# B&R Automation Studio project CombinedLinenCleanA6 (part 2)

#### picd.var
```iecst
VAR
	STEP : UINT;
END_VAR
VAR RETAIN
	PLS : BOOL;
	LASTSTEP : UINT;
END_VAR
VAR
	O_RunMotor : BOOL;
	I_OutgoingFull : BOOL;
	O_OpenSeparator : BOOL;
	ReleasedToIncline : BOOL;
	ReleasedToInclineET : TIME;
	NoBags : BOOL;
	StopInclineET : TIME;
	StopIncline : BOOL;
	I_PaddleInPosition : BOOL;
	BagArriveIncline : BOOL;
	I_ArriveIncline : BOOL;
	TransitWindowClosedET : TIME;
	TransitWindowClosed : BOOL;
	BagReleasedSep : BOOL;
	I_BagAtSep : BOOL;
	I_TrolleyOutAtBott : BOOL;
	I_TrolleyOnIncline : BOOL;
	BagReleased : BOOL;
	mySeq : UINT;
	myIO : UINT;
	myBufferBag : UINT;
	myRelLine : UINT;
	myLine : UINT;
	myLastBag : UINT;
	myFirstBag : UINT;
	myX20IO : UINT;
	I_BagReleasedSep : BOOL;
	TimerAlarm : TON_10ms;
	myRelBag : UINT;
	myIC : UINT;
	DestValid : BOOL;
	myZone : INT;
	SettledAtSep : BOOL;
	SettledAtSepET : UDINT;
	I_BagInSep : BOOL;
	SettledInSep : BOOL;
	SettledInSepET : UDINT;
	BagArrived : BOOL;
END_VAR
```

### Program Logical/Reference/36_picu7 (IEC) - *PICU7 Incline up Empty trolleys

#### picu.ab
```automation-basic
PROGRAM _CYCLIC
	(* cyclic program *)

;Sequence 30 - Primary Incline Conveyor 4 D[900 + mySeq]

;-----------------------------------------
;Revision 1.00 17/04/2007 D.J. First Issue
;-----------------------------------------
mySeq 	= 36
myIO	= 177
myZone	= 0

I_PaddleInPosition		= X[myIO].X01
I_BagAtSep              = X[myIO].X03
I_BagArriveIncline		= X[myIO].X04
I_OutgoingFull			= X[myIO].X05

O_RunMotor 				= FALSE
O_OpenSeparator			= FALSE

;Setup Sequence
;-----------------------
STEP = D[900 + mySeq]
;Setup Pulse contact
PLS = (STEP <> LASTSTEP)
LASTSTEP = STEP

;If no bags on the buffers then stop the motor
NoBags = (STEP = 1) AND NOT I_BagAtSep
TON_10ms(NoBags,2000,StopIncline,StopInclineET)
TON_10ms(I_OutgoingFull,100,OutgoingFull,OutgoingFullET)

O_RunMotor = (NOT OutgoingFull AND NOT StopIncline AND NOT Std.HaltSysZone[myZone] AND (STEP <> 0) AND (STEP <> 2)); AND (STEP <> 2))

IF (STEP = 0) THEN
;	D[900 + mySeq] = 1
ENDIF

;Run Incline until paddle in position
IF (STEP = 1) THEN
	IF (I_PaddleInPosition AND I_BagAtSep AND O_RunMotor) THEN
		D[900 + mySeq] = 2
	ENDIF
ENDIF

;Open Separator 1.5 seconds
;Allow 3 sec for trolley to be detected releasing from separator
TON_10ms((STEP = 2),150,ReleasedToIncline,ReleasedToInclineET)
TON_10ms(ReleasedToIncline,550,TransitWindowClosed,TransitWindowClosedET)
IF (STEP = 2) THEN
	O_OpenSeparator	= NOT ReleasedToIncline
	IF I_BagArriveIncline OR TransitWindowClosed THEN
		D[900 + mySeq] = 3
	ENDIF
	ELSE
	ReleasedToIncline = FALSE
ENDIF

;Check not stpped on paddle
IF (STEP = 3) THEN
	IF NOT I_PaddleInPosition THEN
		D[900 + mySeq] = 1
	ENDIF
ENDIF

Y[34].Y02		= O_RunMotor
Y[myIO].Y06 	= O_OpenSeparator
END_PROGRAM
```

### Program Logical/Reference/38_picu9 (IEC) - *PICU9 Incline up Empty trolleys

#### picu.ab
```automation-basic
PROGRAM _CYCLIC
	(* cyclic program *)

;Sequence 30 - Primary Incline Conveyor 4 D[900 + mySeq]

;-----------------------------------------
;Revision 1.00 17/04/2007 D.J. First Issue
;-----------------------------------------
mySeq 	= 38
myIO	= 179
myZone	= 0

I_PaddleInPosition		= X[myIO].X01
I_BagAtSep              = X[myIO].X03
I_BagArriveIncline		= X[myIO].X04
I_OutgoingFull			= X[myIO].X05

O_RunMotor 				= FALSE
O_OpenSeparator			= FALSE

;Setup Sequence
;-----------------------
STEP = D[900 + mySeq]
;Setup Pulse contact
PLS = (STEP <> LASTSTEP)
LASTSTEP = STEP

;If no bags on the buffers then stop the motor
NoBags = (STEP = 1) AND NOT I_BagAtSep
TON_10ms(NoBags,750,StopIncline,StopInclineET)
TON_10ms(I_OutgoingFull,100,OutgoingFull,OutgoingFullET)

O_RunMotor = (NOT OutgoingFull AND NOT StopIncline AND NOT Std.HaltSysZone[myZone] AND (STEP <> 0) AND (STEP <> 2))

IF (STEP = 0) THEN
	D[900 + mySeq] = 1
ENDIF

;Run Incline until paddle in position
IF (STEP = 1) THEN
	IF (I_PaddleInPosition AND I_BagAtSep AND O_RunMotor) THEN
		D[900 + mySeq] = 2
	ENDIF
ENDIF

;Open Separator 1.5 seconds
;Allow 3 sec for trolley to be detected releasing from separator
TON_10ms((STEP = 2),150,ReleasedToIncline,ReleasedToInclineET)
TON_10ms(ReleasedToIncline,550,TransitWindowClosed,TransitWindowClosedET)
IF (STEP = 2) THEN
	O_OpenSeparator	= NOT ReleasedToIncline
	IF TransitWindowClosed OR I_BagArriveIncline THEN
		D[900 + mySeq] = 3
	ENDIF
	ELSE
	ReleasedToIncline = FALSE
ENDIF

;Check not stpped on paddle
IF (STEP = 3) THEN
	IF NOT I_PaddleInPosition THEN
		D[900 + mySeq] = 1
	ENDIF
ENDIF

Y[34].Y04 		= O_RunMotor
Y[myIO].Y06 	= O_OpenSeparator
END_PROGRAM
```

### Program Logical/Reference/39_picu10 (IEC) - *PICU10 Incline up Empty trolleys

#### picu.ab
```automation-basic
PROGRAM _CYCLIC
	(* cyclic program *)

;Sequence 30 - Primary Incline Conveyor 4 D[900 + mySeq]

;-----------------------------------------
;Revision 1.00 17/04/2007 D.J. First Issue
;-----------------------------------------
mySeq 	= 39
myIO	= 180
myZone	= 2

I_PaddleInPosition		= X[myIO].X01
I_BagAtSep              = X[myIO].X03
I_BagArriveIncline		= X[myIO].X04
I_OutgoingFull			= X[myIO].X05

O_RunMotor 				= FALSE
O_OpenSeparator			= FALSE

;Setup Sequence
;-----------------------
STEP = D[900 + mySeq]
;Setup Pulse contact
PLS = (STEP <> LASTSTEP)
LASTSTEP = STEP

;If no bags on the buffers then stop the motor
NoBags = (STEP = 1) AND NOT I_BagAtSep
TON_10ms(NoBags,3000,StopIncline,StopInclineET)
TON_10ms(I_OutgoingFull,100,OutgoingFull,OutgoingFullET)

O_RunMotor = (NOT OutgoingFull AND NOT StopIncline AND NOT Std.HaltSysZone[myZone] AND (STEP <> 0) AND (STEP <> 2))

IF (STEP = 0) THEN
	;D[900 + mySeq] = 1
ENDIF

;Run Incline until paddle in position
IF (STEP = 1) THEN
	IF (I_PaddleInPosition AND I_BagAtSep AND O_RunMotor) THEN
		D[900 + mySeq] = 2
	ENDIF
ENDIF

;Open Separator 1.5 seconds
;Allow 3 sec for trolley to be detected releasing from separator
TON_10ms((STEP = 2),150,ReleasedToIncline,ReleasedToInclineET)
TON_10ms(ReleasedToIncline,550,TransitWindowClosed,TransitWindowClosedET)
IF (STEP = 2) THEN
	O_OpenSeparator	= NOT ReleasedToIncline
	IF TransitWindowClosed OR I_BagArriveIncline THEN
		D[900 + mySeq] = 3
	ENDIF
	ELSE
	ReleasedToIncline = FALSE
ENDIF

;Check not stpped on paddle
IF (STEP = 3) THEN
	IF NOT I_PaddleInPosition THEN
		D[900 + mySeq] = 1
	ENDIF
ENDIF

Y[34].Y05 		= O_RunMotor
Y[myIO].Y06 	= O_OpenSeparator
END_PROGRAM
```

### Program Logical/Reference/42_picd13 (IEC) - *PICU13 Incline down Empty trolleys

#### picu.ab
```automation-basic
PROGRAM _CYCLIC
	(* cyclic program *)

;Sequence 30 - Primary Incline Conveyor 4 D[900 + mySeq]

;-----------------------------------------
;Revision 1.00 17/04/2007 D.J. First Issue
;-----------------------------------------
mySeq 	= 42
myIO	= 183
myZone	= 3

I_PaddleInPosition		= X[myIO].X01
I_BagAtSep              = X[myIO].X03
I_BagArriveIncline		= X[myIO].X04
I_OutgoingFull			= X[myIO].X05

O_RunMotor 				= FALSE
O_OpenSeparator			= FALSE

;Setup Sequence
;-----------------------
STEP = D[900 + mySeq]
;Setup Pulse contact
PLS = (STEP <> LASTSTEP)
LASTSTEP = STEP

;If no bags on the buffers then stop the motor
NoBags = (STEP = 1) AND NOT I_BagAtSep
TON_10ms(NoBags,2000,StopIncline,StopInclineET)
TON_10ms(I_OutgoingFull,100,OutgoingFull,OutgoingFullET)

O_RunMotor = (NOT OutgoingFull AND NOT StopIncline AND NOT Std.HaltSysZone[myZone] AND (STEP <> 2))

IF (STEP = 0) THEN
	D[900 + mySeq] = 1
ENDIF

;Run Incline until paddle in position
IF (STEP = 1) THEN
	IF (I_PaddleInPosition AND I_BagAtSep AND O_RunMotor) THEN
		D[900 + mySeq] = 2
	ENDIF
ENDIF

;Open Separator 1.5 seconds
;Allow 3 sec for trolley to be detected releasing from separator
TON_10ms((STEP = 2),150,ReleasedToIncline,ReleasedToInclineET)
TON_10ms(ReleasedToIncline,550,TransitWindowClosed,TransitWindowClosedET)
IF (STEP = 2) THEN
	O_OpenSeparator	= NOT ReleasedToIncline
	IF TransitWindowClosed OR I_BagArriveIncline THEN
		D[900 + mySeq] = 3
	ENDIF
	ELSE
	ReleasedToIncline = FALSE
ENDIF

;Check not stpped on paddle
IF (STEP = 3) THEN
	IF NOT I_PaddleInPosition THEN
		D[900 + mySeq] = 1
	ENDIF
ENDIF

Y[23].Y04 		= O_RunMotor
Y[myIO].Y06 	= O_OpenSeparator
END_PROGRAM
```

### Program Logical/Reference/44_picd15 (IEC) - *PICU15 Incline down Empty trolleys

#### picu.ab
```automation-basic
PROGRAM _CYCLIC
	(* cyclic program *)

;Sequence 30 - Primary Incline Conveyor 4 D[900 + mySeq]

;-----------------------------------------
;Revision 1.00 17/04/2007 D.J. First Issue
;-----------------------------------------
mySeq 	= 44
myIO	= 185
myZone	= 3

I_PaddleInPosition		= X[myIO].X01
I_BagAtSep              = X[myIO].X03
I_BagArriveIncline		= X[myIO].X04
I_OutgoingFull			= X[myIO].X05

O_RunMotor 				= FALSE
O_OpenSeparator			= FALSE

;Setup Sequence
;-----------------------
STEP = D[900 + mySeq]
;Setup Pulse contact
PLS = (STEP <> LASTSTEP)
LASTSTEP = STEP

;If no bags on the buffers then stop the motor
NoBags = (STEP = 1) AND NOT I_BagAtSep
TON_10ms(NoBags,2000,StopIncline,StopInclineET)
TON_10ms(I_OutgoingFull,100,OutgoingFull,OutgoingFullET)

O_RunMotor = (NOT OutgoingFull AND NOT StopIncline AND NOT Std.HaltSysZone[myZone] AND (STEP <> 2))

IF (STEP = 0) THEN
	D[900 + mySeq] = 1
ENDIF

;Run Incline until paddle in position
IF (STEP = 1) THEN
	IF (I_PaddleInPosition AND I_BagAtSep AND O_RunMotor) THEN
		D[900 + mySeq] = 2
	ENDIF
ENDIF

;Open Separator 1.5 seconds
;Allow 3 sec for trolley to be detected releasing from separator
TON_10ms((STEP = 2),150,ReleasedToIncline,ReleasedToInclineET)
TON_10ms(ReleasedToIncline,550,TransitWindowClosed,TransitWindowClosedET)
IF (STEP = 2) THEN
	O_OpenSeparator	= NOT ReleasedToIncline
	IF TransitWindowClosed OR I_BagArriveIncline THEN
		D[900 + mySeq] = 3
	ENDIF
	ELSE
	ReleasedToIncline = FALSE
ENDIF

;Check not stpped on paddle
IF (STEP = 3) THEN
	IF NOT I_PaddleInPosition THEN
		D[900 + mySeq] = 1
	ENDIF
ENDIF

Y[23].Y06 		= O_RunMotor
Y[myIO].Y06 	= O_OpenSeparator
END_PROGRAM
```

### Program Logical/Reference/48_49_fbppr (IEC) - *Full bag pressure reliefs buffers before PUPs

#### fb_pr.var
```iecst
VAR CONSTANT
	Dec_C_MaxPressureReliefs : UINT := 2;
END_VAR
VAR RETAIN
	LASTSTEP : ARRAY[0..Dec_C_MaxPressureReliefs] OF UINT;
END_VAR
VAR
	PLS : ARRAY[0..Dec_C_MaxPressureReliefs] OF BOOL;
	STEP : UINT;
	TimerAlarm : ARRAY[0..Dec_C_MaxPressureReliefs] OF TON_10ms;
	mySeq : UINT;
	I_BagAtPR : ARRAY[0..Dec_C_MaxPressureReliefs] OF BOOL;
	n : INT;
	BagSettled : ARRAY[0..Dec_C_MaxPressureReliefs] OF TON_10ms;
	myRelLine : UINT;
	myLastBag : UINT;
	myBag : UINT;
	O_OpenStop : ARRAY[0..Dec_C_MaxPressureReliefs] OF BOOL;
	myOutLine : ARRAY[0..Dec_C_MaxPressureReliefs] OF USINT;
	I_BagReleased : ARRAY[0..Dec_C_MaxPressureReliefs] OF BOOL;
	BagReleased : ARRAY[0..Dec_C_MaxPressureReliefs] OF BOOL;
	myLine : ARRAY[0..Dec_C_MaxPressureReliefs] OF USINT;
	myZone : INT;
	I_BagInSep : ARRAY[0..3] OF BOOL;
	SettledInSep : ARRAY[0..3] OF TON_10ms;
	x : UINT;
	TestIndex : UINT;
	ReleaseValid : ARRAY[0..4] OF BOOL;
END_VAR
```

### Package Logical/Sequences - *GCS Primary 

- Program Logical/Sequences/10ms/zzPrimSearch (IEC) - *Search for ongoing lines using SLAC looking at last bag in transit (no source held here)

### Program Logical/Sequences/10ms/zzStnSer (IEC, version 2.00.0)

#### zzstnser.ab
```automation-basic
;-----------------------------------------------------
;Sorting Station Search Routine - No changes required!
;-----------------------------------------------------

;----------------------------------------
;Version 1.00 19/12/2005 First Issue D.J.
;Version 2.00 03/11/2010 Revised D.J.
;----------------------------------------

PROGRAM _CYCLIC

;Only one Bank / Loading VC can search in a given scan.

Bank = Bank + 1
IF (Bank > Std.MaxStationBanks) THEN
	Bank = 1
ENDIF

;Clear Array
Std.StnsToPurge = FALSE
LOOP n = 0 TO Std.MaxWeighstations DO
	;IF Stn[n].Purge THEN
	;	Std.StnsToPurge = TRUE
	;ENDIF
	BagInList[n] = FALSE
	SearchBagArray[n] = 0
ENDLOOP
TON_10ms(Std.StnsToPurge,100,StartPurge,StartPurgeET) ; use a timer to wait for all purge events to be recieved from trackview

MixCats			= (D[369] > 0)
MixCusts		= (D[366] > 0)	;Allow mixing of customers?
MixProgs		= (D[367] > 0)	;Allow mixing of Programs?

IF MixProgs	 THEN					;IF mixing programs then type must be mixed also.....
	D[368] =  1
ENDIF
MixProgTyp			= (D[368] > 0) 	;Allow mixing of Program Types?

;IF Std.ReversingBelt THEN
;	MaxReverseWeight	= D[370]			;Max weight to reverse..
;ELSE
	;MaxReverseWeight = 0
;ENDIF
;Send Status to Trackview -- BitWise OR to look at all banks

;PurgeOn = (Std.PurgeBank[1].PurgeOn OR Std.PurgeBank[2].PurgeOn OR Std.PurgeBank[3].PurgeOn OR Std.PurgeBank[4].PurgeOn)
;StatusReg = (Std.PurgeBank[1].StationsStatus OR Std.PurgeBank[2].StationsStatus OR Std.PurgeBank[3].StationsStatus OR Std.PurgeBank[4].StationsStatus)
D[360] = PurgeOn
memcpy(ADR(D[371]),ADR(StatusReg),4)
;Used by other sequences that need to check for Line[x].SpaceBIT direct
;eg. Loading VC will look for Enable.Search = 3
Enable.Search = Bank

IF (Bank <= Std.MaxStationBanks) THEN

	IF (Ldg[Bank].Search = 1) THEN

		Ldg[Bank].Found = 0
		Ldg[Bank].Line  = 0

		SearchFound = 0
		SearchLine  = 0

		Stn[0].QTime = 0

		LOOP x = Ldg[Bank].StartStn TO Ldg[Bank].EndStn DO
		;	x = 11
			n = x
			;Std.StnsToPurge = TRUE    ;KEV

			IF (Std.StnsToPurge AND Std.Purging) THEN	;Search through purge Stations to find bags that can be mixed

				IF Bank = 1 THEN
					Break
;					IF NOT TestTim THEN
;						GOTO Debug
;					ENDIF
				ELSE IF Bank = 2 THEN
					Break
				ENDIF
				;Purge doesn;t need to be in x loop so exit if > 1
				EXITIF x > Ldg[Bank].StartStn
				IF StartPurge THEN
					PurgeBatchSize	= 0
					BatchFound = FALSE
					; 1st put all bags to be searched into an array to reduce scanning through all stations bags
					LOOP r = 0 TO Std.MaxWeighstations DO
				;		Std.PurgeBank[Bank].PurgeBatch[r] = 0
					;	IF Stn[r].Purge AND (Stn[r].Weight > 0) AND NOT BagInList[r] AND (r >= Ldg[Bank].StartStn) AND (r <= Ldg[Bank].EndStn)  THEN
				;			SearchBagArray[Std.MaxWeighstations] = Std.StationBagsStart[Bank] + (r-Ldg[Bank].StartStn)
				;			BagInList[r] = TRUE
					;	ENDIF
						;Shuffle array
						LOOP s = Std.MaxWeighstations DOWNTO 1 DO
							IF (SearchBagArray[s-1] = 0) AND (SearchBagArray[s] > 0) THEN
								SearchBagArray[s-1] = SearchBagArray[s]
								SearchBagArray[s] = 0
								EndofBagArray = (s - 1)
							ENDIF
						ENDLOOP
					ENDLOOP
					;LOOP r = 0 TO EndofBagArray DO ; Start Searching through bags
					r = 0 ;Only search through from 1st bag in array as we already know it is to purge
					ReSearch = FALSE
					MisMatchedLoad = FALSE
					SearchIndex = 0
					StartSearch: ;Marker to re-search
					IF ReSearch THEN
						r = SearchIndex
					ENDIF
					LOOP s = 0 TO Std.MaxWeighstations DO
						PurgeBags[s] = 0
					ENDLOOP
					LOOP s = EndofBagArray DOWNTO 0 DO
						myBag_n = SearchBagArray[r]
						myBag_x = SearchBagArray[s]
						MatchCust = FALSE
						MatchCat = FALSE
						MatchProgType = FALSE
						MatchProg = FALSE
						BankValid = TRUE;((myBag_n >= Ldg[Bank].StartStn) AND (myBag_n <= Ldg[Bank].EndStn) AND (myBag_x >= Ldg[Bank].StartStn) AND (myBag_x <= Ldg[0].EndStn))

						;Check customer 1st
						IF (Bag[myBag_n].Cus = Bag[myBag_x].Cus) OR MixCusts THEN
							MatchCust = TRUE
						ENDIF
						IF (Bag[myBag_n].Cat = Bag[myBag_x].Cat) OR MixCats	 THEN
							MatchCat = TRUE
						ENDIF
					;	IF (Bag[myBag_n].Prg = Bag[myBag_x].Prg) OR MixProgs THEN
					;		MatchProg = TRUE
					;	ENDIF
					;	IF (D[2900 + Bag[myBag_n].Prg] = D[2900 + Bag[myBag_x].Prg]) OR MixProgTyp THEN
					;		MatchProgType = TRUE
					;	ENDIF

						MatchBags = (MatchCust AND MatchCat AND MatchProg AND MatchProgType AND BankValid)
						IF MatchBags THEN ; Put bag into another array so they can be best matched by weight
							;PurgeBags[0] = myBag_n
							PurgeBags[Std.MaxWeighstations] = myBag_x
							LOOP t = Std.MaxWeighstations DOWNTO 1 DO
								IF (PurgeBags[t] > 0) AND (PurgeBags[t-1] = 0) THEN
									PurgeBags[t -1] = PurgeBags[t]
									PurgeBags[t] = 0
									PurgeBatchSize	= t
								ENDIF
							ENDLOOP
						ENDIF
					ENDLOOP ; Ony research if no matching bags, and the bag searched is to small for a batch
					IF ((PurgeBatchSize = 1) AND (Bag[PurgeBags[0]].Wgt < MaxReverseWeight)) THEN
						ReSearch = TRUE
						INC SearchIndex
						;Check when all bags have been searched...
						IF (SearchBagArray[SearchIndex] = 0) THEN
							;INC SearchIndex
							;The only bags left cannot be put in the same bag and should be classified as a mixed load.
							MisMatchedLoad = (SearchIndex > 1)
							LOOP y = 0 TO SearchIndex - 1 DO
								PurgeBags[y] = 	SearchBagArray[y]
							ENDLOOP
							PurgeBatchSize = SearchIndex
						ELSE
							GOTO StartSearch
						ENDIF
					ENDIF

					;ENDLOOP
					;Matching bags are in the array Purge Bags. Try to fit into a load?
					;Bag 0 in the array is that master.. This is the data that will go into a bag.. so we will get the batch weight from this program code.
					;Put all bag into wieght order highest first..
					LOOP r = 0 TO 19 DO
						BagInList[r] = FALSE
						PurgeBagsInWgtOrder[r] = 0
					ENDLOOP
					IF (PurgeBatchSize > 0) THEN
						GetStn =  ((PurgeBags[0] - Std.StationBagsStart[Bank]) + 1)
						IF (GetStn < Std.MaxWeighstations) THEN
							MaxBatchWieght = D[4900 + GetStn] ;SP3
						ENDIF
						IF (MaxBatchWieght = 0) OR (MaxBatchWieght <= MaxReverseWeight) THEN
							 MaxBatchWieght = MaxReverseWeight + 100
						ENDIF

						LOOP r = 0 TO (PurgeBatchSize - 1) DO
							BagWgt = 0
							LOOP s = 0 TO (PurgeBatchSize - 1) DO
								IF (Bag[PurgeBags[s]].Wgt > 0) AND (Bag[PurgeBags[s]].Wgt > BagWgt) AND NOT BagInList[s] THEN
									BagWgt = Bag[PurgeBags[s]].Wgt
									BagNum = PurgeBags[s]
									Index = s
								ENDIF
							ENDLOOP
							PurgeBagsInWgtOrder[r] = USINT(BagNum)
							BagInList[Index] = TRUE
						ENDLOOP ;
						IF (MaxBatchWieght > MaxReverseWeight) AND (Bag[PurgeBagsInWgtOrder[0]].Wgt > 0)THEN ; Check no errors in batch sizes.. Reverse all loads if fault
							;Now bags are in weight order make the best by adding the highest values until bag is full
							BatchWeight = 0
							PurgeBagsQty = 0
							;IF (Bag[PurgeBagsInWgtOrder[0]].Wgt  < MaxBatchWieght) THEN
							BatchWeight = Bag[PurgeBagsInWgtOrder[0]].Wgt
							BatchCount = Bag[PurgeBagsInWgtOrder[0]].Cnt
						;	Std.PurgeBank[Bank].PurgeBatch[0] = PurgeBagsInWgtOrder[0]
							;ENDIF
							LOOP r = 1 TO PurgeBatchSize DO ; Start from 1 as index 0 is highest weight so always in the array
								myBag = PurgeBagsInWgtOrder[r]
								IF ((Bag[myBag].Wgt + BatchWeight) <= MaxBatchWieght) THEN
									BatchWeight = Bag[myBag].Wgt + BatchWeight
									BatchCount = Bag[myBag].Cnt + BatchCount
							;		Std.PurgeBank[Bank].PurgeBatch[PurgeBatchSize] = USINT(myBag)
									PurgeBagsQty = PurgeBagsQty + 1
								ENDIF
								;Shuffle down array
								LOOP s = PurgeBatchSize DOWNTO 1 DO
								;	IF (Std.PurgeBank[Bank].PurgeBatch[s] > 0) AND (Std.PurgeBank[Bank].PurgeBatch[s - 1] = 0) THEN
								;		Std.PurgeBank[Bank].PurgeBatch[s - 1] = Std.PurgeBank[Bank].PurgeBatch[s]
								;		Std.PurgeBank[Bank].PurgeBatch[s] = 0
								;	ENDIF
								ENDLOOP
							;	IF (r = PurgeBatchSize) AND (Std.PurgeBank[Bank].PurgeBatch[0] > 0) THEN
							;		BatchFound = TRUE
							;	ENDIF
							EXITIF BatchFound = TRUE
							ENDLOOP
						ENDIF
;					ELSE
;						GOTO ExitPurge ;Invalid purge..
					ENDIF
					IF BatchFound AND NOT MisMatchedLoad THEN ;Bags found;
						IF (BatchWeight >=  MaxReverseWeight) THEN ; Wieght it OK purge into Bag search for destination.

							IF NO THEN
								SearchFound  		= 99
								SearchLine   		= 0;LineSearch[Choice]
								Ldg[Bank].Search   	= 2
							ELSE	;
								;Check line choice 1st to 4th in order if any valid then exit loop
								;StnNum = (Std.PurgeBank[Bank].PurgeBatch[0] - (Std.StationBagsStart[Bank] - Ldg[Bank].StartStn)) ; Get station number from Bag number.
						;		StnCat =  Bag[Std.PurgeBank[Bank].PurgeBatch[0]].Prg

								LineSearch[1]   = D[3000 + StnCat]
								LineSearch[2]   = D[3100 + StnCat]
								LineSearch[3]   = D[3200 + StnCat]
								LineSearch[4]   = D[3300 + StnCat]

								LOOP Choice = 1 TO 4 DO
									LineValid = (D[20 + LineSearch[Choice]] > 0)
									IF (LineSearch[Choice] > 0) AND (Line[LineSearch[Choice]].SpaceBIT >= 1) AND LineValid THEN
										SearchFound  		= 99
										SearchLine   		= LineSearch[Choice]
										Ldg[Bank].Search   	= 2
									ENDIF
									EXITIF (SearchFound > 0)
								ENDLOOP
							ENDIF
						ELSE ; Load/s is to small reverse.

							SearchFound  		= 98
							SearchLine   		= 0
							Ldg[Bank].Search   	= 2
						ENDIF
					ELSE IF MisMatchedLoad THEN
						SearchFound  		= 97
						SearchLine   		= 0
						Ldg[Bank].Search   	= 2
					ENDIF
					IF SearchFound > 90 THEN ;If bags are found remove from purging Q
;						Std.PurgeBank[Bank].PurgeBagQty	= PurgeBagsQty

;						Std.PurgeBank[Bank].PurgeBatchWieght = BatchWeight
;					Std.PurgeBank[Bank].PurgeBatchCount	= BatchCount
;						LOOP r = 0 TO PurgeBagsQty - 1 DO
;							IF (Std.PurgeBank[Bank].PurgeBatch[r] > 0) THEN
;								StnNum = (Std.PurgeBank[Bank].PurgeBatch[r] - (Std.StationBagsStart[Bank] - Ldg[Bank].StartStn))
;								;Stn[StnNum].QTime = 0
;								;Stn[StnNum].Purge = FALSE
;							ENDIF
;						ENDLOOP
					ENDIF
				ENDIF
			ELSE IF ((Stn[n].QTime > 10) AND (Stn[n].QTime > Stn[0].QTime)) THEN

				;Destination has been given to bag by operator check
				LineSearchManual = Stn[n].DestManual

				IF Std.AutoLineAllocation THEN

					;Automatic Line Allocation - Line Space is never checked even if a destiantion has been edited
					SearchFound  		= n
					SearchLine   		= LineSearchManual
					Stn[0].QTime 		= Stn[n].QTime
					Ldg[Bank].Search   	= 2

				ELSE
					;1st 2nd 3rd and 4th Line choices
					LineSearch[1]   = D[4000 + n]
					LineSearch[2]   = D[4100 + n]
					LineSearch[3]   = D[4200 + n]
					LineSearch[4]   = D[4300 + n]

					;Always Search for at least 1 space
					IF (Stn[n].SpacesRequired = 0) THEN
						Stn[n].SpacesRequired = 1
					ENDIF

					;When manual is selected then the 1st 2nd 3rd and 4th are not checked
					IF (LineSearchManual > 0) THEN
						IF (Line[LineSearchManual].SpaceBIT > 0) THEN
							SearchFound  		= n
							SearchLine   		= LineSearchManual
							Stn[0].QTime 		= Stn[n].QTime
							Ldg[Bank].Search   	= 2
						ENDIF
					ELSE
							;Check line choice 1st to 4th in order if any valid then exit loop

						LOOP Choice = 1 TO 4 DO
							;Choice = 1
							LineValid = (D[20 + LineSearch[Choice]] > 0)
							IF (LineSearch[Choice] > 0) AND (Line[LineSearch[Choice]].SpaceBIT >= Stn[n].SpacesRequired) AND LineValid THEN
								SearchFound  		= n
								SearchLine   		= LineSearch[Choice]
								Stn[0].QTime 		= Stn[n].QTime
								Ldg[Bank].Search   	= 2

							ENDIF
							EXITIF (SearchFound > 0)
						ENDLOOP

					ENDIF

				ENDIF ;/AutoLineAllocation

			ENDIF

		ENDLOOP

		ExitPurge:
		IF (Ldg[Bank].Search = 2) THEN
			Ldg[Bank].Found  = SearchFound
			Ldg[Bank].Line   = SearchLine
		ELSE
			Ldg[Bank].Search = 0 ;Failed
		ENDIF

	ENDIF
ENDIF
Debug:

END_PROGRAM
```

### Program Logical/Sequences/10ms/zzCount (IEC) - Counting frames inputs & Piece Weights

#### zzcount.ab
```automation-basic
PROGRAM _CYCLIC
(* cyclic program *)

;Sorting station counting

CountMode 	= D[994]
CountOn		= (CountMode <> 0)
CountPiece 	= (CountMode = 1)
CountBoth	= (CountMode = 2)
CountCount	= (CountMode = 3)

Stn[1].CntInput 	= X[31].X01
Stn[2].CntInput 	= X[31].X02
Stn[3].CntInput 	= X[31].X03
Stn[4].CntInput 	= X[31].X04
Stn[5].CntInput 	= X[32].X01
Stn[6].CntInput 	= X[32].X02
Stn[7].CntInput 	= X[32].X03
Stn[8].CntInput 	= X[32].X04
Stn[9].CntInput 	= X[33].X01
Stn[10].CntInput 	= X[33].X02

LOOP n = 1 TO Std.MaxWeighstations DO

	;Get the category for the station
	StnCat = Bag[200 + n].Cat
	IF ((StnCat < 0) OR (StnCat > Std.MaxCats)) THEN
		StnCat = 0
	ENDIF

	;Read the Category database setting
	StnUsePiece		= (D[2900 + StnCat] > 0)
	StnPieceWgt		= (D[2800 + StnCat])
	;Set mode depending on loading program selection
	StnCountPiece 	= (CountPiece OR (CountBoth AND StnUsePiece))

	IF CountOn THEN
		;Count by input
		CountPLS[n].CLK = (Stn[n].CntInput AND NOT StnCountPiece)
		CountPLS[n] FUB R_TRIG()

		IF CountPLS[n].Q THEN
			Stn[n].Count = (Stn[n].Count + 1)
		ENDIF

		;Count by piece weight
		IF StnCountPiece THEN
			;Calculate the current count by piece weight
			StnGram = (Bag[200 + n].Wgt * 1000)
			IF (StnGram > 0) THEN
				IF (StnPieceWgt > 0) THEN
					;Calc Here
					Items = (StnGram / StnPieceWgt)
					;round up items
					Remainder = SINT(Items MOD 10)
					IF (Remainder > 4) THEN
						ItemsRound = (Items + 10)
					ELSE
						ItemsRound = Items
					ENDIF
					IF ((ItemsRound / 10) < 32767) THEN
						Stn[n].Count = UINT(ItemsRound / 10)
					ELSE
						Stn[n].Count = 32767
					ENDIF
				ELSE
					Stn[n].Count = 0
				ENDIF
			ELSE
				Stn[n].Count = 0
			ENDIF
		ENDIF
	ELSE
		Stn[n].Count = 0
	ENDIF

ENDLOOP

END_PROGRAM
```

### Program Logical/Sequences/10ms/zzStnMix (IEC) - * Station mixing Customer and Categories

#### zzstnmix.ab
```automation-basic
PROGRAM _CYCLIC
;----------------------
;Sorting Station Mixing
;----------------------

;----------------------------------------
;Version 1.00 09/12/2005 D.J. First Issue
;----------------------------------------

;Notes:
;When the operator changes either the Category or Customer of any station then the report should be written.
;If the Customer or Category is set to zero the report will be written for the previous Cat and Cus however
;the previous Cat and Cus will be set to zero. When the Cat or Cus is next changed there will be no report

IF Std.StationReports THEN

	;Special for Mewa only box 1 to 6 are reported on
	LOOP n = 1 TO Std.MaxWeighstations DO

		StnBag = n + (Std.StationBagsStart[1] - 1) ;Assumes all station bags will follow in order

		IF (ReportLoading[n].Cat = 0) THEN

			;Check if Category or Customer have been changed
			CatChanged 	= (Bag[StnBag].Cat <> StnPrev[n].Cat)
			CatValid   	= (StnPrev[n].Cat > 0)

			CusChanged 	= (Bag[StnBag].Cus <> StnPrev[n].Cus)
			CusValid   	= (StnPrev[n].Cus > 0)

			;Check if anything has been added and current weight is not less than the previous
			WgtValue 	= Stn[n].Weight	- INT(StnPrev[n].Wgt)
			WgtValid 	= (WgtValue > 0)

			;Check if anything has been added and current weight is not less than the previous
			CntValue 	= Stn[n].Count - INT(StnPrev[n].Cnt)
			CntValid 	= (CntValue > 0)

			;Ensure valid values as we report on either a weight or count change
			IF (WgtValue < 0) THEN
				WgtValue = 0
			ENDIF

			IF (CntValue < 0) THEN
				CntValue = 0
			ENDIF

			IF ((CatChanged OR CusChanged) AND CusValid AND CatValid AND (WgtValid OR CntValid)) THEN

				ReportLoading[n].Prg = StnPrev[n].Prg		;Program
				ReportLoading[n].Cat = StnPrev[n].Cat		;Category
				ReportLoading[n].Cus = StnPrev[n].Cus		;Customer
				ReportLoading[n].Wgt = UINT(WgtValue)		;Weight
				ReportLoading[n].Cnt = UINT(CntValue)		;Count
				ReportLoading[n].Stn = n         			;Station
				ReportLoading[n].Mcn = 0					;Machine
				ReportLoading[n].Bid = StnPrev[n].Bid		;Bag ID
				ReportLoading[n].Mis = n
				ReportLoading[n].Act = repMix
				ReportLoading[n].Ur1 = 0
				ReportLoading[n].Ur2 = 0
				ReportLoading[n].Rkg = 0

			ENDIF

			;Set Previous to Current even if the Previous values were not valid
			IF (CatChanged OR CusChanged) THEN
				StnPrev[n].Prg = Bag[StnBag].Prg
				StnPrev[n].Cat = Bag[StnBag].Cat
				StnPrev[n].Cus = Bag[StnBag].Cus
				StnPrev[n].Wgt = Stn[n].Weight
				StnPrev[n].Cnt = Stn[n].Count
				StnPrev[n].Bid = Bag[StnBag].Bid
			ENDIF

		ENDIF

	ENDLOOP

ENDIF

END_PROGRAM
```

### Program Logical/Sequences/10ms/zzStatus (IEC) - * System status

#### zzstatus.ab
```automation-basic
PROGRAM _CYCLIC
(* cyclic program *)

;System Status and Halting
;-------------------------

Std.StopSystem 				= (D[100] <> 0)

Std.EStop 					= NOT X[1].X01
Std.MotorOverload   		= NOT X[1].X02
Std.SafetyOn				= X[1].X03
Std.HaltSys					= NOT Std.SafetyOn ;OR Std.StopSystem)

Std.MaxZones 				= 1
Std.FireAlarm				= X[3].X01// ON when the fire alarm is healthy

Std.SafetyOnZone[0]		= Std.SafetyOn AND Std.FireAlarm
Std.SafetyOnZone[1]		= X[1].X03 AND Std.FireAlarm; Gated area for PIC 3,4,5,11 & PP3
Std.SafetyOnZone[2]		= FALSE; Area between belts on soiled pp12, PIC10
Std.SafetyOnZone[3]		= FALSE ;Loading Area
Std.SafetyOnZone[4]		= FALSE;Loading Area Gated + Upstairs storage

LOOP n = 0 TO Std.MaxZones DO
	Std.HaltSysZone[n]=  NOT Std.SafetyOnZone[n]
ENDLOOP

;Std.SafetyOnVC[30]			= TRUE
;Std.HaltSysVC[30]			= NOT Std.SafetyOnVC[30]
;
;Std.SafetyOnVC[2]			= TRUE
;Std.HaltSysVC[2]			= NOT Std.SafetyOnVC[2]

;set to TRUE if not required
LoadingStopped 	= TRUE ;(Bag[220].Prg = 0)
OngoingStopped 	= TRUE ;(Bag[224].Prg = 0)
OffgoingStopped = TRUE ;(Bag[225].Prg = 0)

;If no Bag In Transit and stop requested then set system to stopped D[100] = 2
IF Std.StopSystem THEN
	IF LoadingStopped AND OngoingStopped AND OffgoingStopped THEN
		D[100] = 2
	ENDIF
ENDIF

;Force I/O Enable - Max ? Minutes
ForceEnable = FALSE

tmrForce.IN = ForceEnable
tmrForce.PT = 90000 ;6000 = 1 Minute
tmrForce FUB TON_10ms()

IF ForceEnable AND NOT tmrForce.Q THEN
	D[319] = 1
ELSE
	D[319] = 0
ENDIF

END_PROGRAM
```

### Program Logical/Sequences/10ms/1_clu_1 (IEC, version 1.00.0) - * Loading unit SLU1

#### 3_slu_1Cyclic.ab
```automation-basic
PROGRAM _CYCLIC
	(* cyclic program *)

;--------------------------------
;Sequence 3 - Loading Unit D[903]
;--------------------------------

;Inputs / Ouputs

;Enable.TransferBelt[1]	= FALSE

//I_BagAtBuffer			= X[3].X10
I_BagFrontPast			= X[5].X13
I_BagInLoadingUnit		= X[5].X12
//I_BagOnCarriage         = X[5].X05

//I_ChuteBlocked			= X[3].X14
SwitchedOn			= (D[20] = 1)

O_MoveCompressorUp		= FALSE
O_MoveCompressorDn		= FALSE

O_OpenBufferStop		= FALSE
O_SteadyCylinders		= FALSE
O_OpenStop	 			= FALSE
CAN[1].BagReady         = FALSE

Enable.CVC[2]           = FALSE

O_OpenBufferStop2		= FALSE

Alarm[1].Name 		= 0
Alarm[1].Bag		= 31
Alarm[1].Beacon		= TRUE
Alarm[1].Extra	 	= 0
Alarm[1].Time		= 6000

;Setup Sequence
;--------------
STEP = D[901]
;Setup Pulse contact
PLS = (STEP <> LASTSTEP)
LASTSTEP = STEP

;Alarm
SwitchFault = ((STEP = 1) AND (I_BagFrontPast OR I_BagInLoadingUnit))
;TON_10ms(((NOT PLS) AND (SwitchFault) OR (STEP = 3) OR (STEP = 11)),3000,Alarm[51],AlarmET[51])

IF (STEP = 0) THEN
	;Disabled
ENDIF

;Check for no bag in loading unit
TON_10ms((NOT I_BagFrontPast AND NOT I_BagInLoadingUnit),200,TripsClear,TripsClearET)
IF (STEP = 1) THEN
	IF (NOT CAN[1].UnloadFinished AND SwitchedOn AND TripsClear) THEN
        D[901] = 2
	ENDIF
ENDIF

;Enable CVC2 to Send Bag
IF (STEP = 2) THEN
	Enable.CVC[2] = TRUE
	O_OpenStop	= TRUE
	IF I_BagFrontPast THEN
		D[901] = 3
   	ENDIF
ENDIF

;Bag Settles at loading unit
TON_10ms(I_BagInLoadingUnit,700,SettledAtStop,SettledAtStopET)
IF (STEP = 3) THEN
	Enable.CVC[2] = TRUE	;Must be on until bag is fully in the unit
	IF SettledAtStop THEN
		D[901] = 4
	ENDIF
	Alarm[1].Name = almBagNotArrived
	Alarm[1].Time		= 2000
ENDIF

;Steady bag
TON_10ms((STEP = 4),200,SteadysDown,SteadysDownET)
IF (STEP = 4) THEN
    IF SteadysDown THEN
		D[901] = 5
	ENDIF
ENDIF

;Steady cylinders on from steps 4 - 5
O_SteadyCylinders = ((STEP >= 4) AND (STEP <= 5))

;Move Steady Cylinders down
IF (STEP <> 5) THEN
	Cat 			= 0
	Cus			= 0
	kg			= 0
ENDIF

;Bag Ready to Driers
IF (STEP = 5) THEN
	IF PLS THEN
		Bag[31].Cat = 0
	ENDIF
	CAN[1].BagReady = TRUE
	IF CAN[1].UnloadFinished THEN
		FinishedLoading = TRUE
	ENDIF
	IF (CAN[1].Category > 0) THEN
		Cat 		= uint(CAN[1].Category)
		Cus			= uint(CAN[1].Customer)
		kg			= (CAN[1].Weight * 10)
	ENDIF
	IF FinishedLoading THEN
		Bag[31].Cat = usint(Cat)
		Bag[31].Cus	= Cus
		Bag[31].Wgt	= kg
		D[901] = 6
	ENDIF
ELSE
	FinishedLoading = FALSE
ENDIF

;Allow steadys to go up
TON_10ms((STEP = 6),200,SteadysUp,SteadysUpET)
IF (STEP = 6) THEN
    IF (SteadysUp  AND (Bag[31].Cat > 0))THEN
		D[901] = 7
	ENDIF
ENDIF

;Wait for Enable from CVC1
IF (STEP = 7) THEN
	IF Enable.CLU[1] THEN
		D[901] = 8
	ENDIF
ENDIF

;Release Bag
IF (STEP = 8) THEN
	O_OpenStop = TRUE
	IF NOT Enable.CLU[1] THEN
		D[901] = 1
	ENDIF
	Alarm[1].Name = almBagNotReleased
	Alarm[1].Time		= 2000
ENDIF

;Alarms
TimerAlarm.IN = NOT PLS AND (Alarm[1].Name > 0)
TimerAlarm.PT = Alarm[1].Time
TimerAlarm FUB TON_10ms()
Alarm[1].On = TimerAlarm.Q
Alarm[1].ET = TimerAlarm.ET
;Outputs
;-------

//Y[3].Y10 = O_OpenBufferStop
Y[5].Y12 = O_SteadyCylinders
Y[5].Y13 = O_OpenStop
;YM07 = O_OpenBufferStop2

//Y[3].Y13 = O_MoveCompressorDn

END_PROGRAM
```

#### 3_slu_1.var
```iecst
VAR RETAIN
	STEP : UINT;
	PLS : BOOL;
	LASTSTEP : UINT;
END_VAR
VAR
	EBagSettled : BOOL;
	EBagSettledET : TIME;
	O_OpenStop : BOOL;
	O_SteadyCylinders : BOOL;
	LoadingUnitClear : BOOL;
	LoadingUnitClearET : TIME;
	CompressCount : UINT;
	O_MoveCompressorUp : BOOL;
	SteadysUpET : TIME;
	SteadysUp : BOOL;
	SteadysDown : BOOL;
	SteadysDownET : TIME;
	I_BagAtBuffer : BOOL;
	O_OpenBufferStop : BOOL;
	I_BagInLoadingUnit : BOOL;
	I_BagFrontPast : BOOL;
	SwitchFault : BOOL;
	TimerAlarm : TON_10ms;
	I_CompressorAtTop : BOOL;
	I_CompressorAtBot : BOOL;
	I_CompressorAtMid : BOOL;
	O_MoveCompressorDn : BOOL;
	BagSettledBuffer : BOOL;
	BagSettledBufferET : TIME;
	I_BagAtSVC1Buffer : BOOL;
	O_SVC1BufferOpen : BOOL;
	I_ChuteBlocked : BOOL;
	I_BagOnCarriage : BOOL;
	O_OpenBufferStop2 : BOOL;
	AlarmET : UDINT;
	BagAtBuffer : BOOL;
	BagAtBufferET : UDINT;
	BufferClear : BOOL;
	SwitchedOn : BOOL;
	I_FrontPast : BOOL;
	I_AtStop : BOOL;
	TripsClear : BOOL;
	TripsClearET : UDINT;
	SettledAtStop : BOOL;
	SettledAtStopET : UDINT;
	Cat : INT;
	Cus : INT;
	kg : INT;
	FinishedLoading : BOOL;
END_VAR
```

### Program Logical/Sequences/10ms/2_cvc1 (IEC) - * SVC1 Up from SLU1 & Loading

#### 8_svc1.var
```iecst
VAR
	I_CarrAtTop : BOOL;
	I_CarrAtBottom : BOOL;
END_VAR
VAR RETAIN
	STEP : UINT;
	PLS : BOOL;
END_VAR
VAR
	LASTSTEP : UINT;
	O_MoveCarrUp : BOOL;
	O_OpenCarrStop : BOOL;
	O_MoveCarrDown : BOOL;
	I_BagOnCarr : BOOL;
	O_OpenBuffer : BOOL;
	BagSettledOnCarr : BOOL;
	BagSettledOnCarrET : TIME;
	I_BagReleased : BOOL;
	TimerAlarm : TON_10ms;
	I_CarrAtMiddle : BOOL;
	I_CarrAtWeighing : BOOL;
	I_NoEmptyBag : BOOL;
	I_CollectEmpty : BOOL;
	I_UseAsLoading : BOOL;
	I_UpPushButton : BOOL;
	I_DownPushButton : BOOL;
	Dst : UINT;
	PButton : BOOL;
	SVCRaw : DINT;
	n : UINT;
	ValidCus : BOOL;
	ValidWgt : BOOL;
	O_AlarmLamp : BOOL;
	ValidCat : BOOL;
	Choice : ARRAY[0..4] OF UINT;
	PButtonET : TIME;
	Status : UINT;
	PastMiddleET : TIME;
	PastMiddle : BOOL;
	ValidDst : BOOL;
	I_CarrAtEmptyBagIn : BOOL;
	I_CarrAtEmptyBagOut : BOOL;
	I_BagAtBufferStopLLevel : BOOL;
	I_BagAtEmptyBufferStop : BOOL;
	O_OpenEmptyBufferStop : BOOL;
	O_OpenFullbufferStop : BOOL;
	MoveDownEmptyOut : BOOL;
	O_BufferStop : BOOL;
	AlarmET : UDINT;
	SettledEmptyBuffer : BOOL;
	SettledEmptyBufferET : UDINT;
	SettledOnCarr : BOOL;
	SettledOnCarrET : UDINT;
	EmptyBufferClear : BOOL;
	SettledBuffer : BOOL;
	SettledBufferET : UDINT;
	EmptyDownToEmptyIn : BOOL;
	EmptyDownToEmptyInET : UDINT;
	EmptyDownToEmptyOut : BOOL;
	EmptyDownToEmptyOutET : UDINT;
	EmptyDownToFullIn : BOOL;
	EmptyDownToFullInET : UDINT;
	UpToTop : BOOL;
	UpToTopET : UDINT;
	O_MoveDownEmptyOut : BOOL;
	ReleaseBrake : BOOL;
	MoveDownStep : BOOL;
	MoveUpStep : BOOL;
	HighSpeedTime : UINT;
	TONHighSpeed : TON_10ms;
	HighSpeedDone : BOOL;
	HighSpeedDoneET : TIME;
	O_Point1_4 : BOOL;
	O_Point5 : BOOL;
	StopDelay : BOOL;
	StopDelayET : UDINT;
	TONSteadys : TON_10ms;
	O_CarriageSteadys : BOOL;
	O_MoveUp : BOOL;
	HighSpeedUp : BOOL;
	HighSpeedUpET : UDINT;
	O_MoveDown : BOOL;
	HighSpeedDn : BOOL;
	HighSpeedDnET : UDINT;
	SteadysIn : BOOL;
	SteadysInET : UDINT;
	O_OpenStop : BOOL;
END_VAR
```

#### 8_svc1Cyclic.ab
```automation-basic
PROGRAM _CYCLIC
	(* cyclic program *)

;--------------------------------------------
;Sequence 8 - SVC1 Vertical conveyor 1 D[908]
;--------------------------------------------

;--------------------------------------------
;Sequence 52 - CVC1 Vertical conveyor 1 D[952]
;--------------------------------------------

;Inputs
I_CarrAtTop				= X[4].X09
I_CarrAtBottom			= X[4].X10

I_BagOnCarr				= X[4].X11
I_BagReleased			= X[2].X11

Enable.CLU[1]       = FALSE
O_OpenEmptyBufferStop	= FALSE
O_MoveCarrUp			= FALSE
O_MoveCarrDown			= FALSE
O_OpenCarrStop			= FALSE
O_Point1_4                  = FALSE
 O_CarriageSteadys    = FALSE
O_Point5            = FALSE

//Enable.LU[1]			= FALSE

Alarm[2].Name 				= 0
Alarm[2].Bag				= 32
Alarm[2].Beacon				= TRUE
Alarm[2].Extra				= 0
Alarm[2].Time			  	= 5000

;Setup Sequence
STEP = D[902]
;Setup Pulse contact
PLS = (STEP <> LASTSTEP)
LASTSTEP = STEP

;Alarm
;TON_10ms(((NOT PLS) AND (STEP <> 2) AND (STEP <> 6)AND (STEP <> 10)AND (STEP <> 11)AND (STEP <> 14) AND (STEP <> 16)),3000,Alarm[52],AlarmET[52])

;Sequence
IF (STEP = 0) THEN
	;Disabled
ENDIF

;Move bag from LU to Carriage
IF (STEP = 1) THEN
	Enable.CLU[1] = (I_CarrAtBottom AND NOT I_BagOnCarr)
	IF I_BagOnCarr THEN
		IF (Bag[31].Cat>0) AND (Bag[32].Cat = 0) THEN
			Bag[32] = Bag[31]
			Bag[31] = Bag[0]
		ENDIF
		D[902] = 2
	ENDIF
ENDIF

;skip
IF (STEP = 2) THEN
  		D[902] = 3
 ENDIF

;settle on carriage
TON_10ms((STEP = 3) AND (I_BagOnCarr),300,SettledOnCarr,SettledOnCarrET)
IF (STEP = 3) THEN
	 IF  SettledOnCarr THEN
        D[902] = 4
 	ENDIF
	Alarm[2].Time	= 1500
	Alarm[2].Name 	= almBagNotArrived
ENDIF

;bag settles on carriage
//TON_10ms((I_BagOnCarr),300,SettledOnCarr,SettledOnCarrET)
IF (STEP = 4) THEN
 	O_MoveCarrUp = (NOT I_CarrAtTop)
	IF I_CarrAtTop THEN
 		D[902] = 5
	ENDIF
	;Alarm[2].Time	= 1500
	;Alarm[2].Name 	= almBagNotSettled
 ENDIF

;move carriage down to empty out
IF (STEP = 5) THEN
	IF Line[18].Clear AND (Bag[33].Cat=0) AND (Bag[54].Cat=0) AND NOT I_BagReleased THEN
			C[18]   = 0
			D[902] = 6
	ENDIF
	IF I_BagReleased THEN
			Alarm[2].Time = 20
			Alarm[2].Name = almSwitchFault
	ELSE
		Alarm[2].Name 	= almGeneralSequence
	ENDIF
ENDIF

;check buffer clear
TON_10ms((STEP = 6),100,StopDelay,StopDelayET)
IF (STEP = 6) THEN
	IF PLS THEN
		C[18] = 0
	ENDIF
	O_OpenCarrStop = (I_CarrAtTop AND StopDelay)
		IF (Bag[32].Cat>0) AND (Bag[33].Cat = 0) THEN
			Bag[33] = Bag[32]
			Bag[32] = Bag[0]
		ENDIF
		IF I_BagReleased THEN
			D[902] = 7
		ENDIF
	Alarm[2].Name = almBagNotReleased
	Alarm[2].Time		= 1000
	Alarm[2].Bag				= 33
ENDIF
//ENDIF

;open carriage stop
IF (STEP = 7) THEN
	O_MoveCarrDown = (NOT I_CarrAtBottom)
	;D[43]          = 2
	IF I_CarrAtBottom THEN
		D[902] = 1
	ENDIF
;	Alarm[2].Name 	= almBagNotArrived

;	Alarm[2].Time	= 1500

ENDIF

;IF ((Bag[33].Dst >= 3) AND (Bag[33].Dst <=10) AND Line[18].Full) THEN
	IF ((Bag[33].Cat>0) AND (Bag[54].Cat = 0) AND Line[18].Full) THEN
			Bag[54] = Bag[33]
			Bag[33] = Bag[0]
		ENDIF
;ENDIF

;Inverter Speed Selections
;-------------------------
;High Speed Used For Up		= 50Hz
;Medium Speed Used For Down	= 50Hz

TON_10ms(O_MoveCarrUp  ,1505,HighSpeedUp,HighSpeedUpET) 	;Expected 16.94 seconds @ 591mm/sec
TON_10ms(O_MoveCarrDown,1440,HighSpeedDn,HighSpeedDnET) 	;Expected 16.94 seconds @ 591mm/sec

IF PLS THEN
	IF MoveDownStep AND I_CarrAtTop THEN
		HighSpeedTime = 1440
	ELSE IF MoveUpStep AND I_CarrAtBottom THEN
		HighSpeedTime = 1505
	ELSE
		HighSpeedTime = 0
	ENDIF
ENDIF
IF STEP = 4 THEN
	Y[8].Y01 = (NOT HighSpeedUp)
	Y[8].Y02 = FALSE
ELSE IF (STEP = 7) THEN
	Y[8].Y01 = FALSE
	Y[8].Y02 = (NOT HighSpeedDn)
ELSE
	Y[8].Y01 = FALSE
	Y[8].Y02 = FALSE
ENDIF

;TONHighSpeed.IN = (MoveDownStep OR MoveUpStep)
;TONHighSpeed.PT = HighSpeedTime
;TONHighSpeed FUB TON_10ms()
;HighSpeedDone 	= TONHighSpeed.Q
;HighSpeedDoneET = TONHighSpeed.ET

;Carriage Steady Cylinders
TON_10ms((O_MoveCarrDown OR O_MoveCarrUp),50,SteadysIn,SteadysInET)
O_CarriageSteadys = (NOT O_MoveCarrUp AND NOT O_MoveCarrDown )

;Alarms
TimerAlarm.IN = NOT PLS AND (Alarm[2].Name > 0)
TimerAlarm.PT = Alarm[2].Time
TimerAlarm FUB TON_10ms()
Alarm[2].On = TimerAlarm.Q
Alarm[2].ET = TimerAlarm.ET

;PLC Outputs
;-----------
Y[9].Y01 = (O_MoveCarrUp AND SteadysIn)
Y[9].Y02 = (O_MoveCarrDown AND SteadysIn)
Y[9].Y03 = (Y[9].Y01 OR Y[9].Y02)
Y[9].Y04 = O_OpenCarrStop
Y[9].Y16 = O_CarriageSteadys

;Y[9].Y16 = O_CarriageSteadys

;Inverter Parameters
;2	Min Freq			20Hz
;4	High Speed			50Hz
;5	Medium Speed		50Hz
;7  Acceleration Time	1sec
;8  Deceleration Time	1sec
;9  Electronic O/L		5.00A
;10	DC Injection freq	7Hz
;11 DC Injection Time	1sec
;12	DC Brake Voltage	14%
;13	Starting freq		20Hz
;30	Regenerative fun	1
;42	Output freq detect	0.5Hz
;70	Brake duty			5%
;79 Operation mode		3
;80 Motor capicity 		1.5Kw
;83	Rated motor voltage	400v
;84	Rated motor freq	50Hz

END_PROGRAM
```

### Program Logical/Sequences/10ms/3_cic1 (IEC) - * SPC1 Empty bags up

#### 9_spc1Cyclic.ab
```automation-basic
PROGRAM _CYCLIC
	(* cyclic program *)

;----------------------------------------------
;Sequence 10 - SPC1 Pneumatic Conveyor 1 D[910]
;----------------------------------------------

;Inputs
;Incline Conveyor
;-----------------------------------------
;Revision 1.00 09/01/2002 D.J. First Issue
;-----------------------------------------

I_PaddleinPosition		= X[5].X04
I_BaginIncline			= X[5].X03
//I_BagatBuffer			= X[5].X10

O_RunMotor 				= FALSE
O_OpenBufferStop		= FALSE

Request.CP[5] 			= FALSE

;Setup Sequence
;-----------------------
STEP = D[903]
;Setup Pulse contact
PLS = (STEP <> LASTSTEP)
LASTSTEP = STEP

;Alarm[mySeq].Name 	= 0
Alarm[mySeq].Bag	= 20
Alarm[mySeq].Beacon	= TRUE
Alarm[mySeq].Extra	= 0
Alarm[mySeq].Time	= 3000
;Run Incline until paddle in position
IF (STEP = 1) THEN
	O_RunMotor = (NOT I_PaddleinPosition)
	IF I_PaddleinPosition THEN
		D[903] = 2
	ENDIF
ENDIF

;Check romm in buffer
TON_10ms(I_BagatBuffer,300,BagSettledBuffer,BagSettledBufferET)
IF (STEP = 2) THEN
//	IF (BagSettledBuffer AND (Bag[224].Cat = 0)) THEN
		D[903] = 3
//	ENDIF
ENDIF

;

;Wait for bag in incline
IF (STEP = 3) THEN
Request.CP[5] = TRUE

		IF (Bag[51].Cat>0) AND (Bag[36].Cat=0) THEN
		//		Bag[36] = Bag[51]
		//		Bag[51] = Bag[0]
		ENDIF
	IF I_BaginIncline THEN
		D[903] = 4
	ENDIF
ENDIF

;Let bag settle at base of incline
TON_10ms((STEP = 4),1000,BagSettled,BagSettledET)
IF (STEP = 4) THEN
	IF BagSettled THEN
		D[903] = 5
	ENDIF
ENDIF

;Move Bag up incline
TON_10ms((STEP = 5),200,BagNearTop,BagNearTopET)
IF (STEP = 5) THEN
	O_RunMotor = TRUE
	IF BagNearTop THEN
		D[903] = 6
	ENDIF
ENDIF

;Wait for Ongoing Sequence to Enable
;Run motor for 0.5 seconds
IF (STEP <6) THEN
	O_Select[1] = FALSE
	O_Select[4] = FALSE
	O_Select[2] = FALSE
ENDIF

TON_10ms((STEP = 6),50,RunOn,RunOnET)
IF (STEP = 6) THEN
	O_RunMotor 		= NOT RunOn
	IF (Bag[37].Cat = 0) THEN
		IF (Bag[36].Dst = 1) AND Line[1].Clear AND (Bag[77].Cat=0) THEN
			C[1] = 0
			IF (Bag[36].Cat>0)AND (Bag[37].Cat=0)THEN
				Bag[37] = Bag[36]
				Bag[36] = Bag[0]
			ENDIF
			O_Select[1] = TRUE
			D[903]         = 7
		ELSE IF (Bag[36].Dst = 4) AND Line[4].Clear AND (Bag[72].Cat=0) THEN
			C[4] = 0
			IF (Bag[36].Cat>0)AND (Bag[37].Cat=0)THEN
				Bag[37] = Bag[36]
				Bag[36] = Bag[0]
			ENDIF
			O_Select[4] = TRUE
			D[903]          = 7
		ELSE IF ((Bag[36].Dst = 2) OR  (Bag[36].Dst = 3))AND Line[17].Clear AND (Bag[38].Cat=0) AND NOT Y[9].Y13  THEN
			C[17] = 0
			IF (Bag[36].Cat>0)AND (Bag[37].Cat=0)THEN
				Bag[37] = Bag[36]
				Bag[36] = Bag[0]
			ENDIF
			O_Select[2] = TRUE
			D[903]         = 7
	     ENDIF
	ENDIF
ENDIF

;Run incline until bag at storage lines
IF (STEP = 7) THEN
	O_RunMotor 		= TRUE
	IF (Bag[37].Cat>0)AND (Bag[72].Cat=0)THEN
	//			Bag[72] = Bag[37]
	//			Bag[37] = Bag[0]
	ENDIF
	IF O_Select[1]  THEN
		IF Line[1].Full THEN
			IF (Bag[37].Cat>0)AND (Bag[77].Cat=0)THEN
				Bag[77] = Bag[37]
				Bag[37] = Bag[0]
				Bag[77].Dst = 0
				D[903] = 1
			ENDIF
		ENDIF
	ELSE IF O_Select[4]  THEN
		IF Line[4].Full THEN
			IF (Bag[37].Cat>0)AND (Bag[72].Cat=0)THEN
				Bag[72] = Bag[37]
				Bag[37] = Bag[0]
				Bag[72].Dst = 0
				D[903] = 1
			ENDIF
		ENDIF
	ELSE IF O_Select[2]  THEN
		IF Line[17].Full THEN
			IF (Bag[37].Cat>0)AND (Bag[38].Cat=0)THEN
				Bag[38] = Bag[37]
				Bag[37] = Bag[0]
				D[903] = 1
			ENDIF
		ENDIF
	ENDIF
	;Bag in transit arrives at the buffers

ENDIF

;Alarms
TimerAlarm.IN 		= NOT PLS AND (Alarm[mySeq].Name > 0)
TimerAlarm.PT 		= Alarm[mySeq].Time
TimerAlarm FUB TON_10ms()
Alarm[mySeq].On 	= TimerAlarm.Q
Alarm[mySeq].ET 	= TimerAlarm.ET

Y[9].Y09 = O_RunMotor
Y[6].Y06 = O_Select[1]
//Y[6].Y07 = O_Select[5]
Y[6].Y03 = O_Select[1] OR O_Select[4]
Y[6].Y04 = O_Select[2]
Y[6].Y05 = O_Select[4]
END_PROGRAM
```

### Program Logical/Sequences/10ms/4_cic2 (IEC) - * SPC1 Empty bags up

#### 9_spc1.var
```iecst
VAR
	I_CarrAtTop : BOOL;
	I_CarrAtBottom : BOOL;
END_VAR
VAR RETAIN
	STEP : UINT;
END_VAR
VAR
	PLS : BOOL;
END_VAR
VAR RETAIN
	LASTSTEP : UINT;
END_VAR
VAR
	O_MoveCarrUp : BOOL;
	O_OpenCarrStop : BOOL;
	O_MoveCarrDown : BOOL;
	I_BagOnCarr : BOOL;
	O_OpenBuffer : BOOL;
	SettledBuffer : BOOL;
	SettledBufferET : TIME;
	I_BagAtBuffer : BOOL;
	BagSettledOnCarr : BOOL;
	BagSettledOnCarrET : TIME;
	I_BagReleased : BOOL;
	TimerAlarm : TON_10ms;
	I_BagAtLLBuff : BOOL;
	O_LLBuffOpen : BOOL;
	SettledBufferSDC2ET : TIME;
	SettledBufferSDC2 : BOOL;
	I_BagAtBufferSDC2 : BOOL;
	Alt : USINT;
	O_OpenBuffer1 : BOOL;
	I_PaddleinPosition : BOOL;
	I_BaginIncline : BOOL;
	I_BagatBuffer : BOOL;
	O_RunMotor : BOOL;
	O_OpenBufferStop : BOOL;
	BagSettledBuffer : BOOL;
	BagSettledBufferET : UDINT;
	BagSettled : BOOL;
	BagSettledET : UDINT;
	BagNearTop : BOOL;
	BagNearTopET : UDINT;
	RunOn : BOOL;
	RunOnET : UDINT;
	O_Select : ARRAY[0..6] OF BOOL;
END_VAR
```

#### 9_spc1Cyclic.ab
```automation-basic
PROGRAM _CYCLIC
	(* cyclic program *)

;----------------------------------------------
;Sequence 10 - SPC1 Pneumatic Conveyor 1 D[910]
;----------------------------------------------

;Inputs
;Incline Conveyor
;-----------------------------------------
;Revision 1.00 09/01/2002 D.J. First Issue
;-----------------------------------------

I_PaddleinPosition		= X[5].X06
I_BaginIncline			= X[5].X05
I_BagatBuffer			= X[5].X10

O_RunMotor 				= FALSE
O_OpenBufferStop		= FALSE

Request.CIC[1]			= FALSE

;Setup Sequence
;-----------------------
STEP = D[904]
;Setup Pulse contact
PLS = (STEP <> LASTSTEP)
LASTSTEP = STEP

;Alarm
;TON_10ms(((NOT PLS) AND (STEP = 3)),1000,Alarm[9],AlarmET[9])

;Run Incline until paddle in position
IF (STEP = 1) THEN
	O_RunMotor = (NOT I_PaddleinPosition)
	IF I_PaddleinPosition THEN
		D[904] = 2
	ENDIF
ENDIF

;Check romm in buffer
TON_10ms(I_BagatBuffer,300,BagSettledBuffer,BagSettledBufferET)
IF (STEP = 2) THEN
	IF (BagSettledBuffer AND (Bag[39].Cat = 0) AND (Bag[38].Cat>0)) THEN
		D[904] = 3
	ENDIF
ENDIF

;

;Wait for bag in incline
IF (STEP = 3) THEN
O_OpenBufferStop = TRUE
//	IF I_BaginIncline THEN
		IF (Bag[38].Cat>0) AND (Bag[39].Cat=0) THEN
				Bag[39] = Bag[38]
				Bag[38] = Bag[0]
		ENDIF
	IF I_BaginIncline THEN
		D[904] = 4
	ENDIF
ENDIF

;Let bag settle at base of incline
TON_10ms((STEP = 4),1000,BagSettled,BagSettledET)
IF (STEP = 4) THEN
O_OpenBufferStop = TRUE
	IF BagSettled THEN
		D[904] = 5
	ENDIF
ENDIF

;Move Bag up incline
TON_10ms((STEP = 5),400,BagNearTop,BagNearTopET)
IF (STEP = 5) THEN
O_OpenBufferStop = TRUE
	O_RunMotor = TRUE
	IF BagNearTop THEN
		D[904] = 6
	ENDIF
ENDIF

;Wait for Ongoing Sequence to Enable
;Run motor for 0.5 seconds
IF (STEP <6)THEN
	O_Select[2] = FALSE
	O_Select[3] = FALSE
ENDIF

TON_10ms((STEP = 6),50,RunOn,RunOnET)
IF (STEP = 6) THEN
	O_RunMotor 		= NOT RunOn
	IF (Bag[40].Cat = 0) THEN
		IF (Bag[39].Dst = 2) AND Line[2].Clear AND (Bag[10].Cat=0) THEN
			C[2] = 0
			O_Select[2] = TRUE
			D[904]         = 7
		ELSE IF (Bag[39].Dst = 3) AND Line[3].Clear AND (Bag[13].Cat=0) THEN
			C[3] = 0
			O_Select[3] = TRUE
			D[904]          = 7
		ENDIF
	ENDIF
ENDIF

;Run incline until bag at storage lines
IF (STEP = 7) THEN
	O_RunMotor 		= TRUE
	IF (Bag[40].Dst = 2) THEN
		O_Select[2] = TRUE
	ELSE IF (Bag[40].Dst = 3) THEN
		O_Select[3] = TRUE
	ENDIF
	IF (Bag[39].Cat>0)AND (Bag[40].Cat=0)THEN
				Bag[40] = Bag[39]
				Bag[39] = Bag[0]
	ENDIF
	 IF O_Select[2]  THEN
		IF Line[2].Full THEN
			IF (Bag[40].Cat>0)AND (Bag[10].Cat=0)THEN
				Bag[10] = Bag[40]
				Bag[40] = Bag[0]
				Bag[10].Dst = 0
				D[904] = 1
			ENDIF
		ENDIF
	ELSE IF O_Select[3]  THEN
		IF Line[3].Full THEN
			IF (Bag[40].Cat>0)AND (Bag[13].Cat=0)THEN
				Bag[13] = Bag[40]
				Bag[40] = Bag[0]
				Bag[13].Dst = 0
				D[904] = 1
			ENDIF
		ENDIF

	ENDIF
	;Bag in transit arrives at the buffers

ENDIF

Y[9].Y10 = O_RunMotor
Y[6].Y08 = O_Select[2]
Y[6].Y07 = O_Select[3]
Y[9].Y13 = O_OpenBufferStop

END_PROGRAM
```

### Program Logical/Sequences/10ms/5_cic3 (IEC) - * SPC1 Empty bags up

#### 9_spc1.var
```iecst
VAR
	I_CarrAtTop : BOOL;
	I_CarrAtBottom : BOOL;
END_VAR
VAR RETAIN
	STEP : UINT;
END_VAR
VAR
	PLS : BOOL;
END_VAR
VAR RETAIN
	LASTSTEP : UINT;
END_VAR
VAR
	O_MoveCarrUp : BOOL;
	O_OpenCarrStop : BOOL;
	O_MoveCarrDown : BOOL;
	I_BagOnCarr : BOOL;
	O_OpenBuffer : BOOL;
	SettledBuffer : BOOL;
	SettledBufferET : TIME;
	I_BagAtBuffer : BOOL;
	BagSettledOnCarr : BOOL;
	BagSettledOnCarrET : TIME;
	I_BagReleased : BOOL;
	TimerAlarm : TON_10ms;
	I_BagAtLLBuff : BOOL;
	O_LLBuffOpen : BOOL;
	SettledBufferSDC2ET : TIME;
	SettledBufferSDC2 : BOOL;
	I_BagAtBufferSDC2 : BOOL;
	Alt : USINT;
	O_OpenBuffer1 : BOOL;
	I_PaddleinPosition : BOOL;
	I_BaginIncline : BOOL;
	I_BagatBuffer : BOOL;
	O_RunMotor : BOOL;
	O_OpenBufferStop : BOOL;
	BagSettledBuffer : BOOL;
	BagSettledBufferET : UDINT;
	BagSettled : BOOL;
	BagSettledET : UDINT;
	BagNearTop : BOOL;
	BagNearTopET : UDINT;
	RunOn : BOOL;
	RunOnET : UDINT;
	mySeq : USINT;
	myFirstBag : BOOL;
	O_Select : ARRAY[0..6] OF BOOL;
	ENDI : BOOL;
END_VAR
```

#### 9_spc1Cyclic.ab
```automation-basic
PROGRAM _CYCLIC
	(* cyclic program *)

;----------------------------------------------
;Sequence 10 - SPC1 Pneumatic Conveyor 1 D[910]
;----------------------------------------------

;Inputs
;Incline Conveyor
;-----------------------------------------
;Revision 1.00 09/01/2002 D.J. First Issue
;-----------------------------------------

I_PaddleinPosition		= X[5].X08
I_BaginIncline			= X[5].X07
//I_BagatBuffer			= X[5].X10

O_RunMotor 				= FALSE
O_OpenBufferStop		= FALSE

//Request.SIC[3]			= FALSE
Enable.CDC[2]             = FALSE
Request.CIC[3]            = FALSE
mySeq                          = 5
;-----------------------
STEP = D[905]
;Setup Pulse contact
PLS = (STEP <> LASTSTEP)
LASTSTEP = STEP

;Alarm[mySeq].Name 	= 0
Alarm[mySeq].Bag	= 10016
Alarm[mySeq].Beacon	= TRUE
Alarm[mySeq].Extra	= 0
Alarm[mySeq].Time	= 3000
;Run Incline until paddle in position
IF (STEP = 1) THEN
	O_RunMotor = (NOT I_PaddleinPosition)
	IF I_PaddleinPosition THEN
		D[905] = 2
	ENDIF
ENDIF

;Check romm in buffer
TON_10ms(I_BagatBuffer,300,BagSettledBuffer,BagSettledBufferET)
IF (STEP = 2) THEN
//	IF (BagSettledBuffer AND (Bag[224].Cat = 0)) THEN
		D[905] = 3
//	ENDIF
ENDIF

;

;Wait for bag in incline
IF (STEP = 3) THEN
Enable.CDC[2]  = TRUE
;	IF I_BaginIncline THEN
;		IF (Bag[51].Cat>0) AND (Bag[36].Cat=0) THEN
;				Bag[36] = Bag[51]
;				Bag[51] = Bag[0]
;		ENDIF
	IF I_BaginIncline THEN
		D[905] = 4
	ENDIF
ENDIF

;Let bag settle at base of incline
TON_10ms((STEP = 4),1000,BagSettled,BagSettledET)
IF (STEP = 4) THEN
	IF BagSettled THEN
		D[905] = 5
	ENDIF
ENDIF

;Move Bag up incline
TON_10ms((STEP = 5),200,BagNearTop,BagNearTopET)
IF (STEP = 5) THEN
	O_RunMotor = TRUE
	IF BagNearTop THEN
		D[905] = 6
	ENDIF
ENDIF

;Wait for Ongoing Sequence to Enable
;Run motor for 0.5 seconds
TON_10ms((STEP = 6),50,RunOn,RunOnET)
IF (STEP = 6) THEN
	O_RunMotor 		= NOT RunOn
	Request.CIC[3] = TRUE
	IF Enable.CIC[3] then
		D[905] = 7
	ENDIF
ENDIF

;Run incline until bag at storage lines
IF (STEP = 7) THEN
	O_RunMotor 		= TRUE
		IF NOT Enable.CIC[3] THEN
			D[905] = 1
		ENDIF

	;Bag in transit arrives at the buffers

ENDIF

;Alarms
TimerAlarm.IN 		= NOT PLS AND (Alarm[mySeq].Name > 0)
TimerAlarm.PT 		= Alarm[mySeq].Time
TimerAlarm FUB TON_10ms()
Alarm[mySeq].On 	= TimerAlarm.Q
Alarm[mySeq].ET 	= TimerAlarm.ET

Y[9].Y11 = O_RunMotor

END_PROGRAM
```

### Program Logical/Sequences/10ms/1_stnsa (IEC) - * Honeycombe Stations 1 - 16 - GREEN LAMPS

#### 1_stnsa.var
```iecst
VAR
	n : UINT;
	OpenBag : ARRAY[0..99] OF BOOL;
	STEP : UINT;
	PLS : ARRAY[0..99] OF BOOL;
	LASTSTEP : ARRAY[0..99] OF UINT;
	BagClosed : ARRAY[0..99] OF BOOL;
	BagClosedET : ARRAY[0..99] OF TIME;
	OpenTime : UINT;
	BagOpenedET : ARRAY[0..99] OF TIME;
	BagOpened : ARRAY[0..99] OF BOOL;
	CloseTime : UINT;
	Bank : UINT;
	TimerOpen : ARRAY[0..49] OF TON_10ms;
	TimerClosed : ARRAY[0..49] OF TON_10ms;
	TimerAlarm : ARRAY[0..49] OF TON_10ms;
	StnBag : UINT;
	StnMix : BOOL;
END_VAR
```

#### 1_stnsaCyclic.ab
```automation-basic
PROGRAM _CYCLIC
	(* cyclic program *)

;Honeycombe Sorting Station Control
;----------------------------------------------------
;Revision 1.00 10/01/2002 D.J. First Issue
;Revision 2.00 07/02/2005 D.J. Removed Stn Mix
;Revision 3.00 22/08/2006 D.J. Changed to timer array
;----------------------------------------------------

;Timers
OpenTime  = 700
CloseTime = 300

TON_10ms(    OpenBag[1],OpenTime ,BagOpened[1],BagOpenedET[1])
TON_10ms(NOT OpenBag[1],CloseTime,BagClosed[1],BagClosedET[1])
TON_10ms(    OpenBag[2],OpenTime ,BagOpened[2],BagOpenedET[2])
TON_10ms(NOT OpenBag[2],CloseTime,BagClosed[2],BagClosedET[2])
TON_10ms(    OpenBag[3],OpenTime ,BagOpened[3],BagOpenedET[3])
TON_10ms(NOT OpenBag[3],CloseTime,BagClosed[3],BagClosedET[3])
TON_10ms(    OpenBag[4],OpenTime ,BagOpened[4],BagOpenedET[4])
TON_10ms(NOT OpenBag[4],CloseTime,BagClosed[4],BagClosedET[4])
TON_10ms(    OpenBag[5],OpenTime ,BagOpened[5],BagOpenedET[5])
TON_10ms(NOT OpenBag[5],CloseTime,BagClosed[5],BagClosedET[5])
TON_10ms(    OpenBag[6],OpenTime ,BagOpened[6],BagOpenedET[6])
TON_10ms(NOT OpenBag[6],CloseTime,BagClosed[6],BagClosedET[6])
TON_10ms(    OpenBag[7],OpenTime ,BagOpened[7],BagOpenedET[7])
TON_10ms(NOT OpenBag[7],CloseTime,BagClosed[7],BagClosedET[7])
TON_10ms(    OpenBag[8],OpenTime ,BagOpened[8],BagOpenedET[8])
TON_10ms(NOT OpenBag[8],CloseTime,BagClosed[8],BagClosedET[8])
TON_10ms(    OpenBag[9],OpenTime ,BagOpened[9],BagOpenedET[9])
TON_10ms(NOT OpenBag[9],CloseTime,BagClosed[9],BagClosedET[9])
TON_10ms(    OpenBag[10],OpenTime ,BagOpened[10],BagOpenedET[10])
TON_10ms(NOT OpenBag[10],CloseTime,BagClosed[10],BagClosedET[10])
TON_10ms(    OpenBag[11],OpenTime ,BagOpened[11],BagOpenedET[11])
TON_10ms(NOT OpenBag[11],CloseTime,BagClosed[11],BagClosedET[11])
TON_10ms(    OpenBag[12],OpenTime ,BagOpened[12],BagOpenedET[12])
TON_10ms(NOT OpenBag[12],CloseTime,BagClosed[12],BagClosedET[12])
TON_10ms(    OpenBag[13],OpenTime ,BagOpened[13],BagOpenedET[13])
TON_10ms(NOT OpenBag[13],CloseTime,BagClosed[13],BagClosedET[13])
TON_10ms(    OpenBag[14],OpenTime ,BagOpened[14],BagOpenedET[14])
TON_10ms(NOT OpenBag[14],CloseTime,BagClosed[14],BagClosedET[14])
TON_10ms(    OpenBag[15],OpenTime ,BagOpened[15],BagOpenedET[15])
TON_10ms(NOT OpenBag[15],CloseTime,BagClosed[15],BagClosedET[15])
TON_10ms(    OpenBag[16],OpenTime ,BagOpened[16],BagOpenedET[16])
TON_10ms(NOT OpenBag[16],CloseTime,BagClosed[16],BagClosedET[16])

LOOP n = 1 TO Std.MaxWeighstations DO

	Bag[200+n].Wgt = Stn[n].Weight

	STEP = D[920 + n]
	;Setup Pulse contact
	PLS[n] = (STEP <> LASTSTEP[n])
	LASTSTEP[n] = STEP

	;Step 0 - Disabled
	IF STEP = 0 THEN
		Stn[n].LampOn = TRUE
		Stn[n].CloseFlap = TRUE
		;Disabled
	ENDIF

	IF STEP = 1 THEN
		Stn[n].LampOn = TRUE
		IF D[901] = n THEN
			D[901] = 0
		ENDIF
		IF BagClosed[n] THEN
			D[920 + n] = 2
		ENDIF
	ENDIF

	IF STEP = 2 THEN
		IF D[901] = n THEN
			D[920 + n] = 3
		ENDIF
	ENDIF

	IF STEP = 3 THEN
		Stn[n].LampOn = TRUE
		Stn[n].CloseFlap = TRUE
		;StnMix[n].Cat[0] = 0 ;Set All Mixing Registers to 0 for this station report must have been done
		IF (BagOpened[n] AND ((Stn[n].Weight < 30) OR Test.Stations) AND Ldg[1].BeltHasRun) THEN//Std.TransferBeltRun) THEN
			D[920 + n] = 1
		ENDIF
	ENDIF
	OpenBag[n] = (STEP = 3)

ENDLOOP

;Outputs
;-------

Y[12].Y05 = OpenBag[1]
Y[12].Y06 = OpenBag[2]
Y[12].Y07 = OpenBag[3]
Y[12].Y08 = OpenBag[4]
Y[13].Y05 = OpenBag[5]
Y[13].Y06 = OpenBag[6]
Y[13].Y07 = OpenBag[7]
Y[13].Y08 = OpenBag[8]
Y[14].Y05 = OpenBag[9]
Y[14].Y06 = OpenBag[10]
Y[14].Y07 = OpenBag[11]
Y[14].Y08 = OpenBag[12]
Y[15].Y05 = OpenBag[13]
Y[15].Y06 = OpenBag[14]
Y[15].Y07 = OpenBag[15]
Y[15].Y08 = OpenBag[16]

;Lamps to Outputs - From weighing / search
Y[12].Y01 = (Stn[1].LampOn  OR (Stn[1].LampFlashFast AND Std.Clock100ms))
Y[12].Y02 = (Stn[2].LampOn  OR (Stn[2].LampFlashFast AND Std.Clock100ms))
Y[12].Y03 = (Stn[3].LampOn  OR (Stn[3].LampFlashFast AND Std.Clock100ms))
Y[12].Y04 = (Stn[4].LampOn  OR (Stn[4].LampFlashFast AND Std.Clock100ms))
Y[13].Y01 = (Stn[5].LampOn  OR (Stn[5].LampFlashFast AND Std.Clock100ms))
Y[13].Y02 = (Stn[6].LampOn  OR (Stn[6].LampFlashFast AND Std.Clock100ms))
Y[13].Y03 = (Stn[7].LampOn  OR (Stn[7].LampFlashFast AND Std.Clock100ms))
Y[13].Y04 = (Stn[8].LampOn  OR (Stn[8].LampFlashFast AND Std.Clock100ms))
Y[14].Y01 = (Stn[9].LampOn  OR (Stn[9].LampFlashFast AND Std.Clock100ms))
Y[14].Y02 = (Stn[10].LampOn OR (Stn[10].LampFlashFast AND Std.Clock100ms))
Y[14].Y03 = (Stn[11].LampOn OR (Stn[11].LampFlashFast AND Std.Clock100ms))
Y[14].Y04 = (Stn[12].LampOn OR (Stn[12].LampFlashFast AND Std.Clock100ms))
Y[15].Y01 = (Stn[13].LampOn OR (Stn[13].LampFlashFast AND Std.Clock100ms))
Y[15].Y02 = (Stn[14].LampOn OR (Stn[14].LampFlashFast AND Std.Clock100ms))
Y[15].Y03 = (Stn[15].LampOn OR (Stn[15].LampFlashFast AND Std.Clock100ms))
Y[15].Y04 = (Stn[16].LampOn OR (Stn[16].LampFlashFast AND Std.Clock100ms))

Y[8].Y01 = Stn[1].CloseFlap
Y[8].Y02 = Stn[2].CloseFlap
Y[8].Y03 = Stn[3].CloseFlap
Y[8].Y04 = Stn[4].CloseFlap
Y[8].Y05 = Stn[5].CloseFlap
Y[8].Y06 = Stn[6].CloseFlap
Y[8].Y07 = Stn[7].CloseFlap
Y[8].Y08 = Stn[8].CloseFlap
Y[8].Y09 = Stn[9].CloseFlap
Y[8].Y10 = Stn[10].CloseFlap
Y[8].Y11 = Stn[11].CloseFlap
Y[8].Y12 = Stn[12].CloseFlap
Y[8].Y13 = Stn[13].CloseFlap
Y[8].Y14 = Stn[14].CloseFlap
Y[8].Y15 = Stn[15].CloseFlap
Y[8].Y16 = Stn[16].CloseFlap
END_PROGRAM
```

### Program Logical/Sequences/10ms/2_belt1 (IEC) - * STB1 Transfer Belt 1

#### 2_belt1.var
```iecst
VAR
	MinBeltRunCV : UINT;
	MinBeltRun : BOOL;
	BeltClearET : TIME;
	BeltClear : BOOL;
	LinenDetectedET : TIME;
	LinenDetected : BOOL;
	n : UINT;
	STEP : UINT;
	Step6ET : TIME;
	LASTSTEP : UINT;
	PLS : BOOL;
	O_RunBelt : BOOL;
	RunBelt : BOOL;
	TimerAlarm : TON_10ms;
	I_PhotoBottom : BOOL;
	I_PhotoTop : BOOL;
	Bank : UINT;
	WeightValid : BOOL;
	WeightValue : INT;
	BeltRunTime : UINT;
	BeltAddTime : UINT;
	CountValue : INT;
	CountValid : BOOL;
	StnBag : UINT;
END_VAR
```

#### 2_belt1Cyclic.ab
```automation-basic
PROGRAM _CYCLIC
 	(* cyclic program *)

;Sequence 2 - Transfer Belt 1 from Stations 1-12

;-----------------------------------------
;Revision 1.00 18/01/2006 D.J. First Issue
;-----------------------------------------

;Inputs and Outputs
;------------------

Bank 						= 1

I_PhotoBottom 				= X[5].X14
I_PhotoTop   				= X[5].X14

Request.TransferBelt	= FALSE

O_RunBelt 					= FALSE

Alarm[2].Name 				= 0
Alarm[2].Bag				= 220
Alarm[2].Beacon				= TRUE
Alarm[2].Extra				= 0
Alarm[2].Time				= 5000

n = D[901] ;Selected Station

STEP = D[902]
;Setup Pulse contact
PLS = (STEP <> LASTSTEP)
LASTSTEP = STEP

;Step 0 - Disabled
IF STEP = 0 THEN
	;Disabled
ENDIF

;Step 1 - Check no stations are releasing
IF STEP = 1 THEN
	;Don't allow stations to release
	Ldg[Bank].EnableStnRelease = FALSE
	;No Station Releaseng and switched on
	IF ((D[901] = 0) AND (D[11] > 0)) THEN
		IF (Bag[219].Cat = 0) THEN
			D[902] = 2 ;No Bag on belt
		ELSE
			D[902] = 4 ;Bag on belt
		ENDIF
	ENDIF
	Alarm[2].Name = almNoAlarm
ENDIF

;Step 2 - Enable Station search
IF STEP = 2 THEN

	;Check each station to see if a manual destination has been set
	LOOP n = Ldg[Bank].StartStn TO Ldg[Bank].EndStn DO

		StnBag = n + (Std.StationBagsStart[Bank] - 1)

		IF ((Bag[StnBag].Dst > 0) AND (Bag[StnBag].Dst < 99) AND (D[11] > 0)) THEN ;Dest 99 = Empty Bag in station
			Stn[n].DestManual = Bag[StnBag].Dst
		ELSE
			Stn[n].DestManual = 0
		ENDIF
		;For pairing set number of spaces to search for
		Stn[n].SpacesRequired = 0 ;D[2000 + Bag[StnBag].Prg]

	ENDLOOP

	;Station Search
	IF ((Ldg[Bank].Search = 0) AND (D[11] > 0) AND NOT Std.EStop) THEN
		Ldg[Bank].Search = 1
	ELSE IF ((Ldg[Bank].Search = 2) AND (Ldg[Bank].Found > 0))  THEN

		D[901] 	= Ldg[Bank].Found
		n 		= D[901]

		StnBag 	= n + (Std.StationBagsStart[Bank] - 1)

		;Clear the release button count if used
		Stn[n].ManualRelease 	= FALSE
		Stn[n].PBCount 			= 0

		;------Write Report------
		IF Std.StationReports  THEN

			IF (ReportLoading[n].Cat = 0) THEN

				;Check if anything has been added and current weight is not less than the previous
				WeightValue = Stn[n].Weight - INT(StnPrev[n].Wgt)
				WeightValid = (WeightValue > 0)

				;Check if anything has been added and current weight is not less than the previous
				CountValue = Stn[n].Count - INT(StnPrev[n].Cnt)
				CountValid = (CountValue > 0)

				IF (WeightValid OR CountValid) THEN

					;Ensure valid values as we report on either a weight or count change
					IF (WeightValue < 0) THEN
						WeightValue = 0
					ENDIF

					IF (CountValue < 0) THEN
						CountValue = 0
					ENDIF

		;			ReportLoading[n].Prg = Bag[StnBag].Prg 			;Program
					ReportLoading[n].Cat = Bag[StnBag].Cat			;Category
					ReportLoading[n].Cus = Bag[StnBag].Cus			;Customer
					ReportLoading[n].Wgt = UINT(WeightValue)		;Weight
					ReportLoading[n].Cnt = UINT(CountValue)			;Count
					ReportLoading[n].Stn = n         				;Station
					ReportLoading[n].Mcn = 0						;Machine
				;	ReportLoading[n].Bid = Bag[StnBag].Bid			;Batch ID
				ENDIF

			ENDIF

		ENDIF

		;Set Previous Cat and Cus to Current and Clear Weight and Count
;		StnPrev[n].Prg 	= Bag[StnBag].Prg
		StnPrev[n].Cat 	= Bag[StnBag].Cat
		StnPrev[n].Cus 	= Bag[StnBag].Cus
		StnPrev[n].Wgt 	= 0
		StnPrev[n].Cnt 	= 0
;		StnPrev[n].Bid 	= Bag[StnBag].Bid

		;Copy Station Data to Belt Bag
		Bag[219] 		= Bag[StnBag]			;Copy complete bag data
		Bag[219].Dst 	= USINT(Ldg[Bank].Found)	;Destination
		Bag[StnBag].Dst = 0 					;Reset Destination (Manual)

		;Clear Manual Release and Count
		Stn[n].ManualRelease 	= FALSE
		Stn[n].Count			= 0

		;If Stations are too close to the loading unit then jump to wait for loading unit
		;IF (n >= 1) AND (n <= 4) THEN
		;	D[902] = 6
		;ELSE
			BeltAddTime = (D[901] / 2)
			Ldg[Bank].EnableStnRelease = TRUE
			D[902] = 3
		;ENDIF

		Alarm[2].Name = almNoAlarm

	ENDIF
ELSE
	Ldg[Bank].Search  	= 0 ;Clear Search if not on step 2
ENDIF

;Step 3
;Open Bag and Release to Belt Conveyor
IF STEP = 3 THEN
;	O_RunBelt  = TRUE
;	IF (I_PhotoBottom OR I_PhotoTop	OR Test.TransferBelt) THEN
		D[902] = 4
;	ENDIF
;	Alarm[2].Name = almPhotocellNotMade
ENDIF

;Step 4 - Skipped
IF STEP = 4 THEN
	O_RunBelt = TRUE
	D[902] = 5
	Alarm[2].Name = almNoAlarm
ENDIF

;Step 5 - Run belt until top photocell is made.
IF STEP = 5 THEN
	O_RunBelt = TRUE
	IF I_PhotoTop OR Test.TransferBelt THEN
		D[902] = 6
	ENDIF
;	Alarm[2].Name = almPhotocellNotMade
ENDIF

;Step 6 - Wait for loading unit ready
TON_10ms((STEP = 6),10,RunBelt,Step6ET)
IF STEP = 6 THEN
	O_RunBelt = (NOT RunBelt AND Ldg[Bank].EnableStnRelease)
	IF Enable.TransferBelt THEN
		D[902] = 7
	ENDIF
ENDIF

;Step 7 - Run Belt until linen detected for 1 second and Station has emptied
TON_10ms(((STEP = 7) AND I_PhotoTop),100,LinenDetected,LinenDetectedET)
IF STEP = 7 THEN
	O_RunBelt = TRUE
	Ldg[Bank].EnableStnRelease = TRUE ;Enable Station to Open bags if they haven't been already
	IF (LinenDetected OR Test.TransferBelt) THEN
		D[902] = 8
	ENDIF
;	Alarm[2].Name = almPhotocellNotMade
ENDIF

;Step 8 - Run Belt until photocells clear for 5 seconds
TON_10ms(((STEP = 8) AND NOT I_PhotoBottom AND NOT I_PhotoTop AND NOT Std.EStop),500,BeltClear,BeltClearET)
IF STEP = 8 THEN
	O_RunBelt = TRUE
	IF (BeltClear AND MinBeltRun AND (D[901] = 0)) THEN
		D[902] = 9
	ENDIF
	IF NOT Std.EStop THEN
		IF I_PhotoBottom OR I_PhotoTop THEN
	;		Alarm[2].Name = almPhotocellBlocked
		ELSE IF (D[901] <> 0) THEN
	;		Alarm[2].Name = almStationNotClosed
		ELSE IF NOT MinBeltRun THEN
		;	Alarm[2].Name = almClearingBeltPleaseWait
		ENDIF
	ENDIF
ENDIF

;Note - Unitl the Station has closed the min belt run time won't start
;Note - Speed for Horozintal belt = 45m/min and Inclined 55m/min
BeltRunTime = (10 + BeltAddTime)
CTU((O_RunBelt AND Std.Clock1s AND (D[901] = 0) AND NOT Std.EStop),(STEP = 1),BeltRunTime,MinBeltRun,MinBeltRunCV)

;Step 9 - Check Stations Are Closed
IF STEP = 9 THEN
	;Move Belt bag to loading unit
	IF PLS AND ((Bag[220].Cat = 0) OR (Bag[220].Cat = Std.MaxCats)) AND (Bag[219].Cat > 0) THEN ;OCMW Special!!!!!!!!!
		Bag[220] = Bag[219]
		Bag[219] = Bag[0]
	ENDIF
	IF (D[901] = 0) THEN
		D[902] = 1
	ENDIF
;	Alarm[2].Name = almStationNotClosed
ENDIF

;Alarms
TimerAlarm.IN = NOT PLS AND (Alarm[2].Name > 0)
TimerAlarm.PT = Alarm[2].Time
TimerAlarm FUB TON_10ms()
Alarm[2].On = TimerAlarm.Q
Alarm[2].ET = TimerAlarm.ET

;Outputs
;Inform Station Sequences that the belt has been
Ldg[Bank].BeltHasRun = ((D[902] > 3) AND Ldg[Bank].EnableStnRelease)

Y[10].Y10 = O_RunBelt
END_PROGRAM
```

### Program Logical/Sequences/10ms/3_slu_1 (IEC, version 1.00.0) - * Loading unit SLU1

#### 3_slu_1Cyclic.ab
```automation-basic
PROGRAM _CYCLIC
	(* cyclic program *)

;Sequence 3 - Loading Unit D[903]

;Loading Unit
;--------------------------------------------------------
;Revision 1.00 09/01/2002 D.J. First Issue
;Revision 2.00 15/05/2002 D.J. Added Compression Cylinder
;--------------------------------------------------------

;I_BagAtBuffer			= X712
I_BagSLU1Trip			= X[5].X13
I_BaginLoadingUnit		= X[5].X12
;I_BagOutSLU1			= X714

I_CompressorAtTop		= X[7].X05
I_CompressorAtMid		= X[7].X06
I_CompressorAtBot		= X[7].X07
I_ChuteBlocked			= X[7].X08

O_SteadyCylinders		= FALSE
O_OpenStop	 			= FALSE
O_OpenBuffer 			= FALSE
O_BagSupport			= FALSE
O_Compression			= FALSE

Enable.SVC2				= FALSE

;Setup Sequence
;-----------------------
STEP = D[903]
;Setup Pulse contact
PLS = (STEP <> LASTSTEP)
LASTSTEP = STEP

;Alarm
;TON_10ms(((NOT PLS) AND ((STEP = 3) OR (STEP = 8) OR (STEP = 13))),3000,Alarm[3],AlarmET[3])

;Skipped - Normally Wait for Empty bag at buffer
TON_10ms((NOT I_BagSLU1Trip AND NOT I_BaginLoadingUnit),200,TripsClear,TripsClearET)
IF (STEP = 1) THEN
	IF TripsClear THEN
		D[903] = 2
	ENDIF
ENDIF

;Open stops let bag in Loading Unit
IF (STEP = 2) THEN
	O_OpenStop = TRUE
	IF I_BagSLU1Trip THEN ;bag past stop
		D[903] = 3
	ENDIF
ENDIF

Enable.SVC2 = ((STEP = 2) OR (STEP = 3)) ;Bag must be fully in loading unit before SVC2 can go back up hence STEP = 3

;Wait for bag to settle
TON_10ms(I_BaginLoadingUnit,700,EBagSettled,EBagSettledET)
IF (STEP = 3) THEN
	IF EBagSettled THEN
		D[903] = 4
	ENDIF
ENDIF

;Move Steady Cylinders down
TON_10ms((STEP = 4),300,SCylindersDown,SCylindersDownET)
IF (STEP = 4) THEN
	O_SteadyCylinders 	= TRUE
	O_BagSupport		= TRUE
	IF SCylindersDown THEN
		D[903] = 5
	ENDIF
ENDIF

;Wait for bag to be loaded
IF (STEP = 5) THEN
	O_SteadyCylinders 	= TRUE
	O_BagSupport		= TRUE
	IF I_CompressorAtTop THEN
		Enable.TransferBelt = TRUE
	ENDIF
	IF (Bag[220].Cat > 0) THEN
		IF I_ChuteBlocked THEN
			D[903] = 10				;If the Chute is blocked then go to service routine
		ELSE
			D[903] = 6				;Chute is clear
		ENDIF
	ENDIF
ELSE
	Enable.TransferBelt = FALSE
ENDIF

;Allow Steady Cylinders to move up
TON_10ms((STEP = 6),300,BagSupportDown,BagSupportDownET)
IF (STEP = 6) THEN
	IF BagSupportDown THEN
		D[903] = 7
	ENDIF
ENDIF

;Check svc1 is ready for a bag - If chute is blocked then goto step 10
IF (STEP = 7) THEN
	IF Enable.SLU1 THEN
		D[903] = 8
	ENDIF
ENDIF

;Open stop - unitl bag out
IF (STEP = 8) THEN
	 IF (Bag[220].Cat>0)AND(Bag[221].Cat=0) THEN
						Bag[221] = Bag[220]
						Bag[220] = Bag[0]
		ENDIF                               ;BAGMOVE2(PLS,mem_adr_E,220,221,BagSpacing)
	O_OpenStop = TRUE
	IF NOT Enable.SLU1 THEN
		D[903] = 1
	ENDIF
ENDIF

;Compression Cylinder Service routine
;------------------------------------
TON_10ms((STEP = 10),300,SupportDown,SupportDownET)
IF (STEP = 10) THEN
	O_SteadyCylinders 	= TRUE
	IF SupportDown THEN
		IF NOT I_ChuteBlocked THEN
			D[903] 	= 7	;Chute is clear - goto allow steadys to go up
		ELSE
			D[903] 	= 11 ;Try unblocking chute
			Tries 	= 0
		ENDIF
	ENDIF
ENDIF

;Compress Linen
TON_10ms((STEP = 11),2000,TimedOut,TimedOutET)
IF (STEP = 11) THEN
	O_SteadyCylinders 	= TRUE
	O_Compression 		= TRUE
	IF (I_CompressorAtBot OR TimedOut) THEN
		D[903] = 12
	ENDIF
ENDIF

;Allow compression to go back up
IF (STEP = 12) THEN
	O_SteadyCylinders 	= TRUE
	IF (I_CompressorAtMid OR I_CompressorAtTop) THEN
		IF NOT I_ChuteBlocked THEN
			D[903] 	= 7 	;Chute is clear - goto allow steadys to go up
		ELSE IF (Tries < 5) THEN
			D[903] 	= 11	;Re-try
			Tries	= (Tries + 1)
		ELSE
			D[903]	= 13	;Tried 5 times wait for chute to be cleared
		ENDIF
	ENDIF
ENDIF

;Compression cylinder failed wait for manual clear
IF (STEP = 13) THEN
	O_SteadyCylinders 	= TRUE
	IF (I_CompressorAtMid OR I_CompressorAtTop) THEN
		;IF NOT I_ChuteBlocked THEN
			D[903] 	= 7 	;Chute is clear - goto allow steadys to go up
		;ENDIF
	ENDIF
ENDIF

;Outputs
;-------

Y[5].Y13 = O_OpenStop
;Y711 = O_OpenBuffer
Y[5].Y12 = O_SteadyCylinders
Y[7].Y02 = O_BagSupport
Y[7].Y03 = O_Compression
END_PROGRAM
```

#### 3_slu_1.var
```iecst
VAR RETAIN
	STEP : UINT;
	PLS : BOOL;
	LASTSTEP : UINT;
END_VAR
VAR
	EBagSettled : BOOL;
	EBagSettledET : TIME;
	O_OpenStop : BOOL;
	O_SteadyCylinders : BOOL;
	LoadingUnitClear : BOOL;
	LoadingUnitClearET : TIME;
	I_FullBagOut : BOOL;
	I_CompressorAtBot : BOOL;
	I_CompressorAtMid : BOOL;
	TimerDelayET : TIME;
	O_MoveCompressorDn : BOOL;
	SteadysUpET : TIME;
	SteadysUp : BOOL;
	SteadysDown : BOOL;
	SteadysDownET : TIME;
	I_BagAtBuffer : BOOL;
	I_BagInLoadingUnit : BOOL;
	I_BagFrontPast : BOOL;
	SwitchFault : BOOL;
	TimerAlarm : TON_10ms;
	TimerDelay : BOOL;
	CompressCount : UINT;
	O_MoveCompressorUp : BOOL;
	ElephantsFoot : BOOL;
	I_CompressorAtTop : BOOL;
	I_ChuteBlocked : BOOL;
	BufferClear : BOOL;
	HHHeerR : BOOL;
	I_BagSLU1Trip : BOOL;
	I_BaginLoadingUnit : BOOL;
	O_OpenBuffer : BOOL;
	O_BagSupport : BOOL;
	O_Compression : BOOL;
	AlarmET : UDINT;
	TripsClear : BOOL;
	TripsClearET : UDINT;
	SCylindersDown : BOOL;
	SCylindersDownET : UDINT;
	BagSupportDown : BOOL;
	BagSupportDownET : UDINT;
	SupportDown : BOOL;
	SupportDownET : UDINT;
	Tries : INT;
	TimedOut : BOOL;
	TimedOutET : UDINT;
END_VAR
```

### Program Logical/Sequences/10ms/4_spn1 (IEC) - * Soiled Low  Ongoing Transfer Lines 1 - 6

#### 4_spn1.var
```iecst
VAR
	n : UINT;
END_VAR
VAR RETAIN
	STEP : UINT;
END_VAR
VAR
	ResetPointsET : TIME;
	ResetPoints : BOOL;
	LASTSTEP : UINT;
	PLS : BOOL;
	LineSelect : ARRAY[0..19] OF BOOL;
	OnGoingEnable : BOOL;
	O_Reset : BOOL;
	I_BagatBuffer : ARRAY[0..4] OF BOOL;
	SettledBuffer : ARRAY[0..4] OF BOOL;
	Buffer : UINT;
	AlarmOld : UINT;
	BufferBag : UINT;
	DestValid : BOOL;
	Dest : UINT;
	BufferDst : UINT;
	BufferBagNum : ARRAY[0..4] OF UINT;
	TestBuffer : UINT;
	TimerAlarm : TON_10ms;
	Bfr : UINT;
	BufferSettled : BOOL;
	BufferCat : UINT;
	MaxBuffers : UINT;
	Buff : UINT;
	SettledBufferET : ARRAY[0..4] OF TIME;
	O_OpenSelect : ARRAY[0..4] OF BOOL;
	N : BOOL;
	Reset : BOOL;
END_VAR
```

### Program Logical/Sequences/10ms/5_spf1 (IEC) - * Soiled Offgoing Transfer Lines 1 - 10

#### 5_spf1.var
```iecst
VAR RETAIN
	STEP : UINT;
	LASTSTEP : UINT;
END_VAR
VAR
	PLS : BOOL;
	BagSettledTime : ARRAY[0..99] OF UINT;
	Destination : UINT;
	SettleTime : UINT;
	BestTime : UINT;
	LineSelect : ARRAY[0..49] OF BOOL;
	ResetPointsET : TIME;
	ResetPoints : BOOL;
	n : UINT;
	IncSettle : BOOL;
	LineSettle : ARRAY[0..99] OF BOOL;
	I_BagAtStop : ARRAY[0..49] OF BOOL;
	OffGoingEnable : BOOL;
	AlarmBagNotProx : BOOL;
	SearchDest : UINT;
	TimerAlarm : TON_10ms;
	MaxBuffers : UINT;
	FoundLine : UINT;
	O_Reset : BOOL;
	I_BagReleased : BOOL;
	SDC4_Valid : BOOL;
	SDC1_Valid : BOOL;
	SDC2_Valid : BOOL;
	SDC3_Valid : BOOL;
	BufferBag : ARRAY[0..4] OF UINT;
	BufferClear : ARRAY[0..4] OF BOOL;
	Reset : BOOL;
END_VAR
```

#### 5_spf1Cyclic.ab
```automation-basic
PROGRAM _CYCLIC
	(* cyclic program *)

;----------------------------------------
;Sequence 5 - SPF1 Offgoing Points D[905]
;----------------------------------------
;Inputs
;------

OffGoingEnable 		= ((D[15] > 0) AND NOT Std.HaltSys)

;I_SDCBagAtBuffer[1] = X[6].X01 ;Use for single bag buffer
;I_SDCBagAtBuffer[2] = FALSE ;X[6].X13 ;Use for single bag buffer

;O_SDCBufferOpen[1]  = Y[6].Y01 ;Use for single bag buffer
;O_SDCBufferOpen[2]  = FALSE ;Y[6].Y16 ;Use for single bag buffer

I_BagAtStop[1]  = X[4].X12
I_BagAtStop[2]  = X[4].X13
I_BagAtStop[3]  = X[4].X14
I_BagAtStop[4]  = X[4].X15
I_BagAtStop[5]  = X[4].X16
I_BagAtStop[6]  = X[5].X01
I_BagAtStop[7]  = X[5].X02
I_BagAtStop[8]  = X[5].X03
I_BagAtStop[9]  = X[5].X04
I_BagAtStop[10] = X[5].X05
I_BagAtStop[11] = X[5].X06

;I_BagReleased       = X[14].X03

O_Reset 			= FALSE

;Buffer line configuration
;-------------------------
MaxBuffers			= 2

;BufferBag[1]		= 143 ;Last buffer bag number
;BufferBag[2]		= 151 ;Last buffer bag number

;BufferClear[1] 		= ((D[21] > 0) AND (Bag[190].Cat = 0) AND (Line[21].SpaceBIT > 0) AND (Line[21].Clear))
;BufferClear[2]		= ((D[22] > 0) AND (Bag[190].Cat = 0) AND (Line[22].Space > 0)AND (Line[22].Clear))

Uld[1].SDCReady 	= ((D[16] = 1) AND Line[12].Clear AND NOT Y[3].Y01)
Uld[2].SDCReady 	= ((D[17] = 1) AND Line[13].Clear)
;Passed to unloading search
;Uld[3].SDCReady		= FALSE
;Uld[4].SDCReady 	= FALSE

Alarm[5].Name 		= 0
Alarm[5].Bag		= 190
Alarm[5].Beacon		= TRUE
Alarm[5].Extra		= 0
Alarm[5].Time		= 3000

;Setup Sequence
;--------------
STEP = D[905]
;Setup Pulse contact
PLS = (STEP <> LASTSTEP)
LASTSTEP = STEP

;Sequence Steps
;--------------
IF (STEP = 0) THEN
	;Disabled
ENDIF

;Step 1 - Reset Points
TON_10ms((STEP = 1),300,ResetPoints,ResetPointsET)
IF (STEP = 1) THEN
	O_Reset 	= NOT ResetPoints
	FoundLine 	= 0
	Destination = 0
	IF (ResetPoints AND OffGoingEnable) THEN
		D[905] = 2
	ENDIF
ENDIF

;Bags on storage line timers
R_TRIG(Std.Clock100ms,IncSettle)
AlarmBagNotProx 	= FALSE
AlarmBagNotProxLine = 0

LOOP n = 1 TO Std.MaxLines DO

	LineSettle[n]  = (I_BagAtStop[n] AND (Bag[Line[n].FirstBag].Cat > 0))
	IF IncSettle AND LineSettle[n] AND (BagSettledTime[n] < $FFFF) THEN
		BagSettledTime[n] = BagSettledTime[n] + 1
	ELSE IF NOT LineSettle[n] THEN
		BagSettledTime[n] = 0
		;If Bag has destiantion and not at stop then alarm
		IF (STEP = 2) AND (Bag[Line[n].FirstBag].Dst > 0) THEN
			Alarm[5].Name	= almBagNotAtProx
			Alarm[5].Bag	= Line[n].FirstBag
			Alarm[5].Extra 	= n
		ENDIF
	ENDIF

ENDLOOP

;Buffer trip not correct alarms
LOOP n = 1 TO MaxBuffers DO
	IF (STEP = 2) AND BufferClear[n] AND NOT Uld[n].SDCReady THEN
		Alarm[5].Name 	= almSwitchFault
		Alarm[5].Bag	= BufferBag[n]
	ENDIF
ENDLOOP

;Search for the bag with a valid destination that has been waiting the longest
IF STEP = 2 THEN

	FoundLine 	= 0
	Destination = 0
	BestTime 	= 0
	SettleTime = 30 ;3 seconds

	LOOP n = 1 TO Std.MaxLines DO

		IF (BagSettledTime[n] > SettleTime) THEN
			SearchDest = Bag[Line[n].FirstBag].Dst

			SDC1_Valid  = ((SearchDest = 12) AND Uld[1].SDCReady)
			SDC2_Valid 	= ((SearchDest = 13) AND Uld[2].SDCReady)
			;SDC3_Valid 	= ((SearchDest = 13) AND Uld[3].SDCReady)
			;SDC4_Valid 	= ((SearchDest = 14) AND Uld[4].SDCReady)

			IF (SDC1_Valid OR SDC2_Valid OR SDC3_Valid OR SDC4_Valid) THEN
				FoundLine 	= n
				Destination = SearchDest
				BestTime 	= BagSettledTime[n]
			ENDIF
		ENDIF

	ENDLOOP

	IF ((FoundLine > 0) AND OffGoingEnable AND (Bag[226].Cat = 0) AND Line[Destination].Clear AND (Bag[226].Cat = 0) AND NOT I_BagReleased) THEN
		C[Destination]  = 0
		D[905] = 3
	ENDIF

ENDIF

;Step 3 - Select Line / Open Stop, Until Bag at correct destination
;Clear Line Selections
LOOP n = 1 TO Std.MaxLines DO
	LineSelect[n] = FALSE
ENDLOOP

IF (STEP = 3) THEN

	;Show bag in transit
	IF (Bag[226].Cat = 0) AND (Bag[Line[FoundLine].FirstBag].Cat > 0)THEN
		Bag[226] 						= Bag[Line[FoundLine].FirstBag]
		Bag[Line[FoundLine].FirstBag] 	= Bag[0]
	ENDIF

	IF PLS THEN
			;C[13] = 0
		ENDIF

	;Select Line - Wait for bag to arrive
	LineSelect[FoundLine] = TRUE

	;Select Route
	;IF (I_BagReleased  AND (Bag[Line[13].LastBag].Cat = 0)) THEN
		 ;Unloading Program
	IF (Destination = 12) AND Line[Destination].Trip THEN
		Uld[1].DischargerStartLine = FoundLine
		Bag[227] = Bag[226]
		Bag[226] = Bag[0]
		D[905] 					= 1
	ELSE IF (Destination = 13) AND Line[Destination].Trip THEN
		Uld[2].DischargerStartLine = FoundLine
		Bag[230] = Bag[226]
		Bag[226] = Bag[0]
		D[905] 					= 1
	ENDIF

	Alarm[5].Name	= almBagNotReleased

ENDIF

;move transit bag to buffer
;IF (Bag[190].Cat > 0) AND Line[13].Trip AND (Bag[193].Cat = 0) AND NOT PLS THEN
;	Bag[193] = Bag[190]
;	Bag[190] = Bag[0]
;ENDIF

;Alarms
TimerAlarm.IN = NOT PLS AND (Alarm[5].Name > 0)
TimerAlarm.PT = Alarm[5].Time
TimerAlarm FUB TON_10ms()
Alarm[5].On = TimerAlarm.Q
Alarm[5].ET = TimerAlarm.ET

;Outputs
;-------
Y[5].Y07 = Reset
Y[4].Y12 = LineSelect[1]
Y[4].Y13 = LineSelect[2]
Y[4].Y14 = LineSelect[3]
Y[4].Y15 = LineSelect[4]
Y[4].Y16 = LineSelect[5]
Y[5].Y01 = LineSelect[6]
Y[5].Y02 = LineSelect[7]
Y[5].Y03 = LineSelect[8]
Y[5].Y04 = LineSelect[9]
Y[5].Y05 = LineSelect[10]
Y[5].Y06 = LineSelect[11]
;Y000 = LineSelect[12]
;Y000 = LineSelect[13]
;Y000 = LineSelect[14]

Y[5].Y09 = (D[36] = 1)
Y[5].Y08 = (D[36] = 2)

;Buffer line selection
;Y[4].Y15 = (Destination = 11)
;Y[4].Y16 = (Destination = 12)
;Y[40].Y07 = (Destination = 22)
;Y[40].Y08 = (Destination = 21)
END_PROGRAM
```

### Program Logical/Sequences/10ms/6_sdc1 (IEC) - * SDC1 Machine 1 BCD/CAN

#### 6_sdc1Cyclic.ab
```automation-basic
PROGRAM _CYCLIC
	(* cyclic program *)

;Sequence 6 - Discharger 1 D[906]
a

;-----------------------------------------
;Revision 1.00 19/12/2005 D.J. First Issue
;-----------------------------------------

DischargerEnable 		= ((D[16] > 0) AND NOT Std.HaltSys)

//I_BagAtBuffer			  = X[3].X02
I_BagAtDischarger = X[3].X01
I_SafetyRunning       = X[8].X15

I_OpenBag				= X[6].X15 OR TestDrop           ;X[23].X01
//I_LoadDropped			= CAN[1].LoadDropped OR TestDischarger  ;X[23].X02

O_Steadys				= FALSE ;Y[6].Y01
O_OpenBuffer 			= FALSE ;Y[6].Y02
O_OpenBag				= FALSE ;Y[6].Y03
O_OpenStop				= FALSE ;Y[6].Y04
O_Closer				= FALSE ;Y[6].Y05
O_BagReady          = FALSE

Request.CDC[1] = FALSE

;Alarm
Alarm[6].Name 			= 0 ;Clear sequence alarm name
Alarm[6].Bag 			= 42
Alarm[6].Beacon			= TRUE
Alarm[6].Extra			= 0
Alarm[6].Time			= 3000

;Setup Sequence
STEP = D[906]
;Setup Pulse contact
PLS = (STEP <> LASTSTEP)
LASTSTEP = STEP

;Step 0 - Disabled
IF (STEP = 0) THEN
	;Disabled
ENDIF

;Check Status - Bag settled at buffer, no bag at discharger, bag at buffer on screen and no bag at discharger on the screen
//TON_10ms(I_BagAtBuffer,300,SettledAtBuffer,SettledAtBufferET)
IF (STEP = 1) THEN
	IF  NOT I_BagAtDischarger AND (Bag[42].Cat = 0)  THEN
		D[906] = 2
	ENDIF
	IF (Bag[42].Cat > 0) THEN
		Alarm[6].Name = almBagDataError
	ELSE IF I_BagAtDischarger THEN
		Alarm[6].Name = almSwitchFault
	ENDIF
ENDIF

;Wait for bag in discharger
IF (STEP = 2) THEN
	Request.CDC[1] 	= TRUE
	Enable.CDC4Empty 	= TRUE
	IF I_BagAtDischarger THEN
		D[906] = 3
	ENDIF
	Alarm[6].Name = almBagNotArrived
ENDIF

;Let bag settle in discharger
TON_10ms(((STEP = 3) AND I_BagAtDischarger),1000,SettledAtDischarger,SettledAtDischargerET)
IF (STEP = 3) THEN
	IF (Bag[228].Cat = 0) AND (Bag[227].Cat > 0) THEN
		Bag[228] = Bag[227]
		Bag[227] = Bag[0]
	ENDIF
	IF SettledAtDischarger THEN
		D[906] = 4
	ENDIF
	Alarm[6].Name = almBagNotSettled
ENDIF

;Allow steadys to move down
TON_10ms((STEP = 4),400,SteadysDown,SteadysDownET)
IF (STEP = 4) THEN
	IF SteadysDown AND (Bag[42].Cat <> Std.MaxCats)  THEN
		D[906] = 5
	ENDIF
	IF (Bag[42].Cat = Std.MaxCats) AND SteadysDown THEN
		D[906] = 8
	ENDIF
ENDIF

;Steady cylinders on from steps 4 - 9
O_Steadys = ((STEP >= 4) AND (STEP <= 9))

;Bag opener on from step 5 - 8
O_OpenBag = ((STEP >= 6) AND (STEP <= 8))

;Wash Codes
;IF (STEP = 4) OR (STEP = 5) THEN
;
;;round up weight to give to wash machine
;	Remainder = SINT(Bag[228].Wgt MOD 10)
;	IF (Remainder > 4) THEN
;		WgtRound = (Bag[228].Wgt + 10)
;	ELSE
;		WgtRound = Bag[228].Wgt
;	ENDIF
;
;
;;Codes to CBW
;	CAN[1].Category = Bag[228].Cat
;	CAN[1].Customer = Bag[228].Cus
;	CAN[1].Weight   = (WgtRound / 10)
;ELSE
;	CAN[1].Category = 0
;	CAN[1].Customer = 0
;	CAN[1].Weight   = 0
;ENDIF

;Bag Ready to Washing Machine
IF (STEP = 5) THEN
	O_BagReady = TRUE
	IF I_OpenBag OR TestDischarger THEN
		D[906] = 6
	ENDIF

ENDIF

;Open Bag Until LoadDropped recieved and has been open for 6 seconds
TON_10ms((STEP = 6),600,MinOpen,MinOpenET) ;ET means Elapsed Time
IF (STEP = 6) THEN
	IF (NOT I_OpenBag AND MinOpen) THEN
		D[906] = 7
	ENDIF
	Alarm[6].Name = almLoadNotDropped
ENDIF

;Change display to empty bag
IF (STEP = 7) THEN
	O_BagReady = Std.Clock500ms
	IF ( I_OpenBag  OR TestDrop) THEN ;AND I_BagEmpty) OR TestDrop) THEN
		Bag[42].Cat 	= Std.MaxCats
		D[906] 			= 8
	ENDIF
	Alarm[6].Name = almGeneralSequence
ENDIF

;Close bag
TON_10ms((STEP = 8),700,CloserDown,CloserDownET)
IF (STEP = 8) THEN
	O_Closer = TRUE
	IF CloserDown THEN
		D[906] = 9
	ENDIF
ENDIF

;Allow closer to go back up
TON_10ms((STEP = 9),700,CloserUp,CloserUpET)
IF (STEP = 9) THEN
	IF CloserUp THEN
		D[906] = 10
	ENDIF
ENDIF

;Allow steadys to go up
TON_10ms((STEP = 10),400,SteadyUp,SteadyUpET)
IF (STEP = 10) THEN
	IF SteadyUp THEN
		D[906] = 11
	ENDIF
ENDIF

;Check for space on empty bag buffer
IF (STEP = 11) THEN
 //Request.CDC[1] = TRUE
	IF Enable.CDC[1] THEN
		D[906] = 12
	ENDIF
	ELSE

ENDIF

;Open buffer stop - unitl bag out
IF (STEP = 12) THEN
	O_OpenStop = TRUE
	IF PLS THEN
		;C[14] = 0
	ENDIF
	Bag[42].Cat = 0
	Bag[42].Cus = 0
	Bag[42].Wgt = 0
	IF NOT Enable.CDC[1] THEN
		D[906] = 1
	ENDIF
	Alarm[6].Name = almBagNotReleased
ENDIF

;Alarms
TimerAlarm.IN 	= NOT PLS AND (Alarm[6].Name > 0)
TimerAlarm.PT 	= Alarm[6].Time
TimerAlarm FUB TON_10ms()
Alarm[6].On 	= TimerAlarm.Q
Alarm[6].ET 	= TimerAlarm.ET

;Outputs

Y[3].Y01 = O_BagReady
Y[3].Y01 = O_Steadys
Y[3].Y02 = O_OpenBag
Y[3].Y03 = O_OpenStop
Y[3].Y04 = O_Closer

END_PROGRAM
```

### Program Logical/Sequences/10ms/7_sdc2 (IEC) - * SDC1 Machine 1 BCD/CAN

#### 6_sdc1.var
```iecst
VAR RETAIN
	STEP : UINT;
	PLS : BOOL;
	LASTSTEP : UINT;
	SteadyUp : BOOL;
	CloserUpET : TIME;
	SteadysDown : BOOL;
	SteadysDownET : TIME;
	LoadDropped : BOOL;
END_VAR
VAR
	SteadyUpET : TIME;
	CloserDownET : TIME;
	SettledAtDischargerET : TIME;
	MinOpenET : TIME;
	SettledAtDischarger : BOOL;
	CloserDown : BOOL;
	MinOpen : BOOL;
	CloserUp : BOOL;
	SettledAtBuffer : BOOL;
	SettledAtBufferET : TIME;
	I_BagAtBuffer : BOOL;
	O_OpenStop : BOOL;
	O_OpenBag : BOOL;
	O_Steadys : BOOL;
	O_OpenBuffer : BOOL;
	O_Closer : BOOL;
	I_BagAtDischarger : BOOL;
	I_OpenBag : BOOL;
	I_LoadDropped : BOOL;
	TestDrop : BOOL;
	DischargerEnable : BOOL;
	TestDischarger : BOOL;
	Remainder : SINT;
	TimerAlarm : TON_10ms;
	WgtRound : UINT;
	a : BOOL;
	I_BagEmpty : BOOL;
	I_SafetyRunning : BOOL;
	O_BagReady : BOOL;
END_VAR
```

#### 6_sdc1Cyclic.ab
```automation-basic
PROGRAM _CYCLIC
	(* cyclic program *)

;Sequence 6 - Discharger 1 D[906]
a

;-----------------------------------------
;Revision 1.00 19/12/2005 D.J. First Issue
;-----------------------------------------

DischargerEnable 		= ((D[22] > 0) AND NOT Std.HaltSys)

I_BagAtBuffer			  = X[3].X04
I_BagAtDischarger = X[3].X03
I_SafetyRunning       = X[8].X15

I_OpenBag				= X[7].X15 OR TestDrop           ;X[23].X01
I_LoadDropped			= X[7].X13 OR TestDischarger  ;X[23].X02
I_BagEmpty              = X[2].X13

O_Steadys				= FALSE ;Y[6].Y01
O_OpenBuffer 			= FALSE ;Y[6].Y02
O_OpenBag				= FALSE ;Y[6].Y03
O_OpenStop				= FALSE ;Y[6].Y04
O_Closer				= FALSE ;Y[6].Y05
O_BagReady          = FALSE

;Alarm
Alarm[7].Name 			= 0 ;Clear sequence alarm name
Alarm[7].Bag 			= 43
Alarm[7].Beacon			= TRUE
Alarm[7].Extra			= 0
Alarm[7].Time			= 3000

;Setup Sequence
STEP = D[907]
;Setup Pulse contact
PLS = (STEP <> LASTSTEP)
LASTSTEP = STEP

;Step 0 - Disabled
IF (STEP = 0) THEN
	;Disabled
ENDIF

;Check Status - Bag settled at buffer, no bag at discharger, bag at buffer on screen and no bag at discharger on the screen
TON_10ms(I_BagAtBuffer,300,SettledAtBuffer,SettledAtBufferET)
IF (STEP = 1) THEN
	IF DischargerEnable AND SettledAtBuffer AND  NOT I_BagAtDischarger AND (Bag[43].Cat = 0) AND (Bag[6].Cat > 0)THEN
		D[907] = 2
	ENDIF
	IF (Bag[43].Cat > 0) THEN
		Alarm[7].Name = almBagDataError
	ELSE IF I_BagAtDischarger THEN
		Alarm[7].Name = almSwitchFault
	ENDIF
ENDIF

;Wait for bag in discharger
IF (STEP = 2) THEN
	O_OpenBuffer 	= TRUE
	IF (Bag[43].Cat = 0) AND (Bag[6].Cat>0) THEN
		Bag[43] = Bag[6]
		Bag[6]   = Bag[0]
	ENDIF
	IF I_BagAtDischarger THEN
		D[907] = 3
	ENDIF
	Alarm[7].Name = almBagNotArrived
ENDIF

;Let bag settle in discharger
TON_10ms(((STEP = 3) AND I_BagAtDischarger),1000,SettledAtDischarger,SettledAtDischargerET)
IF (STEP = 3) THEN
;	IF (Bag[228].Cat = 0) AND (Bag[227].Cat > 0) THEN
;		Bag[228] = Bag[227]
;		Bag[227] = Bag[0]
;	ENDIF
	IF SettledAtDischarger THEN
		D[907] = 4
	ENDIF
	Alarm[7].Name = almBagNotSettled
ENDIF

;Allow steadys to move down
TON_10ms((STEP = 4),400,SteadysDown,SteadysDownET)
IF (STEP = 4) THEN
	IF SteadysDown AND (Bag[43].Cat <> Std.MaxCats)  THEN
		D[907] = 5
	ENDIF
	IF (Bag[43].Cat = Std.MaxCats) AND SteadysDown THEN
		D[907] = 8
	ENDIF
ENDIF

;Steady cylinders on from steps 4 - 9
O_Steadys = ((STEP >= 4) AND (STEP <= 9))

;Bag opener on from step 5 - 8
O_OpenBag = ((STEP >= 6) AND (STEP <= 8))

;Wash Codes
;IF (STEP = 4) OR (STEP = 5) THEN
;
;;round up weight to give to wash machine
;	Remainder = SINT(Bag[228].Wgt MOD 10)
;	IF (Remainder > 4) THEN
;		WgtRound = (Bag[228].Wgt + 10)
;	ELSE
;		WgtRound = Bag[228].Wgt
;	ENDIF
;
;
;;Codes to CBW
;	CAN[1].Category = Bag[228].Cat
;	CAN[1].Customer = Bag[228].Cus
;	CAN[1].Weight   = (WgtRound / 10)
;ELSE
;	CAN[1].Category = 0
;	CAN[1].Customer = 0
;	CAN[1].Weight   = 0
;ENDIF

;Bag Ready to Washing Machine
IF (STEP = 5) THEN
	O_BagReady = TRUE
	O_Closer        = TRUE
	IF I_OpenBag OR TestDischarger THEN
		D[907] = 6
	ENDIF

ENDIF

;Open Bag Until LoadDropped recieved and has been open for 6 seconds
TON_10ms((STEP = 6),600,MinOpen,MinOpenET) ;ET means Elapsed Time
IF (STEP = 6) THEN
	IF I_LoadDropped THEN
		LoadDropped = TRUE
	ENDIF
	IF (LoadDropped AND MinOpen) THEN
		D[907] = 7
	ENDIF
	Alarm[7].Name = almLoadNotDropped
	ELSE
	LoadDropped = FALSE
ENDIF

;Change display to empty bag
IF (STEP = 7) THEN
	//O_BagReady = Std.Clock500ms
	IF (NOT I_OpenBag  OR TestDrop) THEN ;AND I_BagEmpty) OR TestDrop) THEN
		Bag[43].Cat 	= Std.MaxCats
		D[907] 			= 8
	ENDIF
	Alarm[7].Name = almGeneralSequence
ENDIF

;Close bag
TON_10ms((STEP = 8),700,CloserDown,CloserDownET)
IF (STEP = 8) THEN
	O_Closer = TRUE
	IF CloserDown THEN
		D[907] = 9
	ENDIF
ENDIF

;Allow closer to go back up
TON_10ms((STEP = 9),700,CloserUp,CloserUpET)
IF (STEP = 9) THEN
	IF CloserUp THEN
		D[907] = 10
	ENDIF
ENDIF

;Allow steadys to go up
TON_10ms((STEP = 10),400,SteadyUp,SteadyUpET)
IF (STEP = 10) THEN
	IF SteadyUp THEN
		D[907] = 11
	ENDIF
ENDIF

;Check for space on empty bag buffer
IF (STEP = 11) THEN

	IF Enable.CDC[2] OR (D[905] = 3) THEN
		D[907] = 12
	ENDIF
	ELSE
	//	Request.CDC[1] = FALSE
ENDIF

;Open buffer stop - unitl bag out
IF (STEP = 12) THEN
	O_OpenStop = TRUE
	IF PLS THEN
		;C[14] = 0
	ENDIF
	Bag[43].Cat = 0
	Bag[43].Cus = 0
	Bag[43].Wgt = 0
	IF (D[905] <>3) THEN
		D[907] = 1
	ENDIF
	Alarm[7].Name = almBagNotReleased
ENDIF

;Alarms
TimerAlarm.IN 	= NOT PLS AND (Alarm[7].Name > 0)
TimerAlarm.PT 	= Alarm[7].Time
TimerAlarm FUB TON_10ms()
Alarm[7].On 	= TimerAlarm.Q
Alarm[7].ET 	= TimerAlarm.ET

;Outputs

Y[3].Y05 = O_OpenBuffer
Y[3].Y06 = O_Steadys
Y[3].Y07 = O_OpenBag
Y[3].Y08 = O_OpenStop
Y[3].Y09 = O_Closer

END_PROGRAM
```

### Program Logical/Sequences/10ms/8_sdc3 (IEC) - * SDC1 Machine 1 BCD/CAN

#### 6_sdc1.var
```iecst
VAR RETAIN
	STEP : UINT;
	PLS : BOOL;
	LASTSTEP : UINT;
	SteadyUp : BOOL;
	CloserUpET : TIME;
	SteadysDown : BOOL;
	SteadysDownET : TIME;
	LoadDropped : BOOL;
END_VAR
VAR
	SteadyUpET : TIME;
	CloserDownET : TIME;
	SettledAtDischargerET : TIME;
	MinOpenET : TIME;
	SettledAtDischarger : BOOL;
	CloserDown : BOOL;
	MinOpen : BOOL;
	CloserUp : BOOL;
	SettledAtBuffer : BOOL;
	SettledAtBufferET : TIME;
	I_BagAtBuffer : BOOL;
	O_OpenStop : BOOL;
	O_OpenBag : BOOL;
	O_Steadys : BOOL;
	O_OpenBuffer : BOOL;
	O_Closer : BOOL;
	I_BagAtDischarger : BOOL;
	I_OpenBag : BOOL;
	I_LoadDropped : BOOL;
	TestDrop : BOOL;
	DischargerEnable : BOOL;
	TestDischarger : BOOL;
	Remainder : SINT;
	TimerAlarm : TON_10ms;
	WgtRound : UINT;
	a : BOOL;
	I_BagEmpty : BOOL;
	MySeq : USINT;
	I_SafetyRunning : BOOL;
	O_BagReady : BOOL;
END_VAR
```

#### 6_sdc1Cyclic.ab
```automation-basic
PROGRAM _CYCLIC
	(* cyclic program *)

;Sequence 6 - Discharger 1 D[906]
a

;-----------------------------------------
;Revision 1.00 19/12/2005 D.J. First Issue
;-----------------------------------------

DischargerEnable 		= ((D[23] > 0) AND NOT Std.HaltSys)
MySeq                       = 8

I_BagAtBuffer			  = X[3].X08
I_BagAtDischarger = X[3].X07
//I_SafetyRunning       = X[8].X15

I_OpenBag				= X[3].X10 OR TestDrop           ;X[23].X01
//I_LoadDropped			= X[7].X13 OR TestDischarger  ;X[23].X02
//I_BagEmpty              = X[2].X13

O_Steadys				= FALSE ;Y[6].Y01
O_OpenBuffer 			= FALSE ;Y[6].Y02
O_OpenBag				= FALSE ;Y[6].Y03
O_OpenStop				= FALSE ;Y[6].Y04
O_Closer				= FALSE ;Y[6].Y05
O_BagReady          = FALSE

;Alarm
Alarm[MySeq].Name 			= 0 ;Clear sequence alarm name
Alarm[MySeq].Bag 			= 44
Alarm[MySeq].Beacon			= TRUE
Alarm[MySeq].Extra			= 0
Alarm[MySeq].Time			= 3000

;Setup Sequence
STEP = D[900+MySeq]
;Setup Pulse contact
PLS = (STEP <> LASTSTEP)
LASTSTEP = STEP

;Step 0 - Disabled
IF (STEP = 0) THEN
	;Disabled
ENDIF

;Check Status - Bag settled at buffer, no bag at discharger, bag at buffer on screen and no bag at discharger on the screen
TON_10ms(I_BagAtBuffer,300,SettledAtBuffer,SettledAtBufferET)
IF (STEP = 1) THEN
	IF DischargerEnable AND SettledAtBuffer AND  NOT I_BagAtDischarger AND (Bag[44].Cat = 0) AND (Bag[11].Cat > 0)THEN
		D[900+MySeq] = 2
	ENDIF
	IF (Bag[44].Cat > 0) THEN
		Alarm[MySeq].Name = almBagDataError
	ELSE IF I_BagAtDischarger THEN
		Alarm[MySeq].Name = almSwitchFault
	ENDIF
ENDIF

;Wait for bag in discharger
IF (STEP = 2) THEN
	O_OpenBuffer 	= TRUE
	IF (Bag[44].Cat = 0) AND (Bag[11].Cat>0) THEN
		Bag[44] = Bag[11]
		Bag[11]   = Bag[0]
	ENDIF
	IF I_BagAtDischarger THEN
		D[900+MySeq] = 3
	ENDIF
	Alarm[7].Name = almBagNotArrived
ENDIF

;Let bag settle in discharger
TON_10ms(((STEP = 3) AND I_BagAtDischarger),1000,SettledAtDischarger,SettledAtDischargerET)
IF (STEP = 3) THEN
;	IF (Bag[228].Cat = 0) AND (Bag[227].Cat > 0) THEN
;		Bag[228] = Bag[227]
;		Bag[227] = Bag[0]
;	ENDIF
	IF SettledAtDischarger THEN
		D[900+MySeq] = 4
	ENDIF
	Alarm[MySeq].Name = almBagNotSettled
ENDIF

;Allow steadys to move down
TON_10ms((STEP = 4),400,SteadysDown,SteadysDownET)
IF (STEP = 4) THEN
	IF SteadysDown AND (Bag[43].Cat <> Std.MaxCats)  THEN
		D[900+MySeq] = 5
	ENDIF
	IF (Bag[43].Cat = Std.MaxCats) AND SteadysDown THEN
		D[900+MySeq] = 8
	ENDIF
ENDIF

;Steady cylinders on from steps 4 - 9
O_Steadys = ((STEP >= 4) AND (STEP <= 9))

;Bag opener on from step 5 - 8
O_OpenBag = ((STEP >= 6) AND (STEP <= 8))

;Wash Codes
;IF (STEP = 4) OR (STEP = 5) THEN
;
;;round up weight to give to wash machine
;	Remainder = SINT(Bag[228].Wgt MOD 10)
;	IF (Remainder > 4) THEN
;		WgtRound = (Bag[228].Wgt + 10)
;	ELSE
;		WgtRound = Bag[228].Wgt
;	ENDIF
;
;
;;Codes to CBW
;	CAN[1].Category = Bag[228].Cat
;	CAN[1].Customer = Bag[228].Cus
;	CAN[1].Weight   = (WgtRound / 10)
;ELSE
;	CAN[1].Category = 0
;	CAN[1].Customer = 0
;	CAN[1].Weight   = 0
;ENDIF

;Bag Ready to Washing Machine
IF (STEP = 5) THEN
	O_BagReady = TRUE
	O_Closer        = TRUE
	IF I_OpenBag OR TestDischarger THEN
		D[900+MySeq] = 6
	ENDIF

ENDIF

;Open Bag Until LoadDropped recieved and has been open for 6 seconds
TON_10ms((STEP = 6),600,MinOpen,MinOpenET) ;ET means Elapsed Time
IF (STEP = 6) THEN
	IF I_OpenBag THEN
		LoadDropped = TRUE
	ENDIF
	IF (NOT I_OpenBag AND MinOpen) THEN
		D[900+MySeq] = 7
	ENDIF
	Alarm[MySeq].Name = almLoadNotDropped
	ELSE
	LoadDropped = FALSE
ENDIF

;Change display to empty bag
IF (STEP = 7) THEN
	IF I_OpenBag THEN
		LoadDropped = TRUE
	ENDIF
	IF (LoadDropped  OR TestDrop) THEN ;AND I_BagEmpty) OR TestDrop) THEN
		Bag[44].Cat 	= Std.MaxCats
		D[900+MySeq] 			= 8
	ENDIF
	Alarm[MySeq].Name = almGeneralSequence
	ELSE
	LoadDropped = FALSE
ENDIF

;Close bag
TON_10ms((STEP = 8),700,CloserDown,CloserDownET)
IF (STEP = 8) THEN
	O_Closer = TRUE
	IF CloserDown THEN
		D[900+MySeq] = 9
	ENDIF
ENDIF

;Allow closer to go back up
TON_10ms((STEP = 9),700,CloserUp,CloserUpET)
IF (STEP = 9) THEN
	IF CloserUp THEN
		D[900+MySeq] = 10
	ENDIF
ENDIF

;Allow steadys to go up
TON_10ms((STEP = 10),400,SteadyUp,SteadyUpET)
IF (STEP = 10) THEN
	IF SteadyUp THEN
		D[900+MySeq] = 11
	ENDIF
ENDIF

;Check for space on empty bag buffer
IF (STEP = 11) THEN
 	Request.CDC[3] = TRUE
	IF Enable.CDC[3]  THEN
		D[900+MySeq] = 12
	ENDIF
	ELSE
		Request.CDC[3] = FALSE
ENDIF

;Open buffer stop - unitl bag out
IF (STEP = 12) THEN
	O_OpenStop = TRUE
	IF PLS THEN
		;C[14] = 0
	ENDIF
	Bag[44].Cat = 0
	Bag[44].Cus = 0
	Bag[44].Wgt = 0
	IF NOT Enable.CDC[3]  THEN
		D[900+MySeq] = 1
	ENDIF
	Alarm[MySeq].Name = almBagNotReleased
ENDIF

;Alarms
TimerAlarm.IN 	= NOT PLS AND (Alarm[MySeq].Name > 0)
TimerAlarm.PT 	= Alarm[MySeq].Time
TimerAlarm FUB TON_10ms()
Alarm[MySeq].On 	= TimerAlarm.Q
Alarm[MySeq].ET 	= TimerAlarm.ET

;Outputs

Y[3].Y10 = O_OpenBuffer
Y[3].Y11 = O_Steadys
Y[3].Y12 = O_OpenBag
Y[3].Y13 = O_OpenStop
Y[3].Y14 = O_Closer
Y[3].Y15 = O_BagReady
END_PROGRAM
```

### Program Logical/Sequences/10ms/9_sdc4 (IEC) - * SDC1 Machine 1 BCD/CAN
